// TIA Portal project "TFM_DanielBejar_S71500_Final" (V17)

(* hardware
DEVICE "S7-1500/ET200MP station_1"  S7-1500 station
   slot 0: "Rail_0"  Rack  6ES7 590-1***0-0AA0
   slot 0: "PS 25W 24VDC_1"  PS 25W 24VDC  6ES7 505-0KA00-0AB0  V1.0
   slot 1: "PLC_1"  CPU 1515-2 PN  6ES7 515-2AM02-0AB0  V2.9
      slot 3: "CPU display_1"  6ES7591-1BA00-0AA0
      slot 32768: "PROFINET interface_1"  X1
         slot 32769: "Port_1"  X1 P1
         slot 32770: "Port_2"  X1 P2
      slot 33024: "PROFINET interface_2"  X2
      slot 34817: "Virtual CP interface port_1"  Virtual CP interface port  Virtual CP interface port
   slot 2: "DI 32x24VDC BA_1"  DI 32x24VDC BA  6ES7 521-1BL10-0AA0  V1.1
   slot 3: "DQ 16x24VDC/0.5A BA_1"  DQ 16x24VDC/0.5A BA  6ES7 522-1BH10-0AA0  V1.1
DEVICE "HMI_1"  TP1200 Comfort
   slot 0: "HMI_1"  TP1200 Comfort  6AV2 124-0MC01-0AX0  17.0.0.0
   slot 1: "HMI_RT_1"  TP1200 Comfort  6AV2 124-0MC01-0AX0  17.0.0.0
   slot 5: "HMI_1.IE_CP_1"  PROFINET Interface  17.0.0.0
      slot 1: "PROFINET Interface_1"  PROFINET Interface
         slot 1: "Port_1"  Port
         slot 2: "Port_2"  Port
   slot 7: "HMI_1.MPI/DP_CP_1"  MPI/DP Interface  17.0.0.0
*)

// ===== PLC "PLC_1"  CPU 1515-2 PN =====

VAR_GLOBAL   // PLC tag table "Default tag table"
   "Clock_Byte" AT %MB255 : Byte;
   "Clock_10Hz" AT %M255.0 : Bool;
   "Clock_5Hz" AT %M255.1 : Bool;
   "Clock_2.5Hz" AT %M255.2 : Bool;
   "Clock_2Hz" AT %M255.3 : Bool;
   "Clock_1.25Hz" AT %M255.4 : Bool;
   "Clock_1Hz" AT %M255.5 : Bool;
   "Clock_0.625Hz" AT %M255.6 : Bool;
   "Clock_0.5Hz" AT %M255.7 : Bool;
END_VAR

VAR_GLOBAL   // PLC tag table "Estados"
   "Estado0" AT %M0.0 : Bool;
   "Estado1" AT %M0.1 : Bool;
   "Estado2" AT %M0.2 : Bool;
   "Estado3" AT %M0.3 : Bool;
   "Estado4" AT %M0.4 : Bool;
   "Estado5" AT %M0.5 : Bool;
   "Estado6" AT %M0.6 : Bool;
   "Estado7" AT %M0.7 : Bool;
   "Estado8" AT %M1.0 : Bool;
   "Estado9" AT %M1.1 : Bool;
   "Estado10" AT %M1.2 : Bool;
   "Estado11" AT %M1.3 : Bool;
   "Estado12" AT %M1.4 : Bool;
   "Estado13" AT %M1.5 : Bool;
   "EstadoPausa" AT %M1.6 : Bool;
   "EstadoError" AT %M1.7 : Bool;
   "Estados" AT %MD0 : DWord;
END_VAR

VAR_GLOBAL   // PLC tag table "IO_Programa"
   "SP_Cintas" AT %EW0 : Word;   // Cada bit se activará según los SP del final de las cintas de materiales
   "ActivacionCintas" AT %AW0 : Word;   // Cada bit indica la activación de una de las cintas
   "CintaGeneral" AT %A1.6 : Bool;   // Activación de la cinta general
   "SP_CintaGeneral" AT %E1.6 : Bool;   // Sensor de presencia de la cinta general
   "ReiniciarSistema" AT %E2.0 : Bool;   // Solicitud desde pulsador de reiniciar sistema
   "SP_CintaEmpaquetado" AT %E1.7 : Bool;   // Sensor de presencia de la cinta de empaquetado
   "CintaEmpaquetado" AT %A1.7 : Bool;   // Activación de la cinta de empaquetado
   "HMI_SP_Cintas" AT %MW10 : Word;   // Entrada simulada del HMI
   "HMI_SP_CintaGeneral" AT %M11.6 : Bool;   // Entrada simulada del HMI
   "HMI_SP_CintaEmpaquetado" AT %M11.7 : Bool;   // Entrada simulada del HMI
   "HMI_PaleE" AT %M12.0 : Bool;   // Entrada simulada del HMI
   "HMI_PaleF" AT %M12.1 : Bool;   // Entrada simulada del HMI
   "HMI_ReiniciarSistema" AT %M12.2 : Bool;   // Reiniciar el sistema desde HMI
END_VAR

DATA_BLOCK "TCP_vbes"   // DB6
{ S7_Optimized_Access := 'FALSE' }
VERSION : 0.1
   VAR
      RX : Array[0..49] of Char;   // Array del mensaje de entrada (RX)
      TX : Array[0..49] of Char;   // Array del mensaje de salida (TX)
      DesconectarServidor : Bool;   // Señal para desconectar el servidor
      TX_Enviar : Bool;   // Señal para enviar el mensaje en TX
      TX_Procesando : Bool;   // Hasta no recibir el ACK, esta vbe será true
      RX_Recibir : Bool := true;   // Habilita la recepción de mensajes
      RX_Procesar : Bool;   // Cuando se recibe un mensaje, se manda a procesar
      TX_Len : UDInt;   // Longitud mensaje TX
      RX_Len : UDInt;   // Longitud mensaje RX
      LastID : Char;   // Ultimo mensaje mandado (para comprobar el ACK)
      TiempoTX : Time;   // Tiempo del sistema cuando se mandó el último TX
      TiempoRX : Time;   // Tiempo del sistema cuando se recibió el último RX
   END_VAR
BEGIN
END_DATA_BLOCK

DATA_BLOCK "SISTEMA_vbes"   // DB8
{ S7_Optimized_Access := 'FALSE' }
VERSION : 0.1
   VAR
      Mesa : Array[0..15] of Word;   // Los bits de Mesa indican si el componente está presente o no en la posición de esa mesa
      Prioridad : Array[0..15] of Int;   // A menor sea el índice, mayor prioridad tiene dicha mesa. Almacena el número de mesa
      Material_Destino : Word;   // Material que será transportado por la cinta general
      Mesa_Destino : Int;   // Mesa en la que irá el material que circula por la cinta general
      Material_EnProceso : Word;   // Variable temporal que almacena el material que el robot está colocando
      Mesa_EnProceso : Int;   // Variable temporal que almacena la mesa que el robot está utilizando
      Mascaras_Cintas : Word;   // Deshabilita un SP de la cinta de materiales. Ocurre cuando el material no es necesario
      NumeroMesas : Word := 4;   // Número de mesas reales en el sistema (máximo 16)
      SP_Enmascarados : Word;   // Los sensores de presencia tras tener en cuenta cuáles están deshabilitados
      IndicePrioridad : Int;   // Indice de la matriz de prioridades
      MatsNecesarios : Word;   // Inversa del contenido en Mesa[]
      SP_Prioritarios : Word;   // Los bits de esta vbe indican si el alimento está disponible y es necesario para la mesa prioritaria
      NumeroMateriales : Int := 5;   // Numero de materiales sin contar caja y tapa
      RobotOcupado : Bool;   // True si el robot está realizando alguna operación
      RobotConectado : Bool;   // True si la conexión con el robot es correcta
      MsgError : String;   // Almacena el último mensaje que ha causado un error
      ElementoBase : Word := 16#20;   // El identificador de la base es bit(NumMateriales)
      ElementoTapa : Word := 16#40;   // El identificador de la tapa es bit(NumMateriales+1)
      ModoSimulacion : Bool;   // Determina si el modo simulación está activo o no
      TActivacionCintaEmp : Time;   // Tiempo hasta el que debe mantenerse activa la cinta de empaquetado
      EstadoAnterior : Word;   // Almacena el estado anterior, sirve para retomar el funcionamiento tras un fallo leve
   END_VAR
BEGIN
   Prioridad[0] := 0;
   Prioridad[1] := 1;
   Prioridad[2] := 2;
   Prioridad[3] := 3;
   Prioridad[4] := 4;
   Prioridad[5] := 5;
   Prioridad[6] := 6;
   Prioridad[7] := 7;
   Prioridad[8] := 8;
   Prioridad[9] := 9;
   Prioridad[10] := 10;
   Prioridad[11] := 11;
   Prioridad[12] := 12;
   Prioridad[13] := 13;
   Prioridad[14] := 14;
   Prioridad[15] := 15;
END_DATA_BLOCK

DATA_BLOCK "HMI_vbes"   // DB9
{ S7_Optimized_Access := 'FALSE' }
VERSION : 0.1
   VAR
      HMI_NumeroMesaSeleccionada : Int;
      HMI_ValorMesaSeleccionada : Word;
      HMI_MesaSeleccionada : Bool;
      HMI_BaseSeleccionada : Bool;
      HMI_TapaSeleccionada : Bool;
      HMI_NumeroMesasDeseadas : Int := 4;
      HMI_NumeroMaterialesDeseados : Int := 5;
      HMI_MostrarPiezaE : Bool;
      HMI_MostrarPiezaF : Bool;
      HMI_MaterialDestino : Word;
      HMI_MesaDestino : Word;
      HMI_Errores : Word;
      HMI_MandarHome : Bool;
      HMI_ApagarRobot : Bool;
      HMI_PausarSistema : Bool;
      HMI_SistemaPausado : Bool;
   END_VAR
BEGIN
END_DATA_BLOCK

// folder: System blocks/Program resources

DATA_BLOCK "TCP_COMMS_DB"   // DB1
{ S7_Optimized_Access := 'TRUE' }
VERSION : 0.1
// stored: InstanceOfName TCP_COMMS
"TCP_COMMS"
BEGIN
END_DATA_BLOCK

DATA_BLOCK "DB_ParamsConexion"   // DB2
{ S7_Optimized_Access := 'TRUE' }
AUTHOR : SIMATIC
FAMILY : MC7Plus
NAME : TC_IP_v4
VERSION : 1.0
// stored: InstanceOfName TCON_IP_v4
"TCON_IP_v4"
BEGIN
   ID := 1;
   InterfaceId := 64;
   RemotePort := 2000;
   ActiveEstablished := true;
   RemoteAddress.ADDR[1] := 192;
   RemoteAddress.ADDR[2] := 168;
   RemoteAddress.ADDR[4] := 130;
END_DATA_BLOCK

// folder: (top level)

FUNCTION_BLOCK "TCP_COMMS"   // FB1, LAD
TITLE = Bloque de comunicaciones TCP
{ S7_Optimized_Access := 'TRUE' }
VERSION : 0.1
// Este bloque está encargado de conectar, desconectar, enviar y recibir mensajes por el puerto TCP. El PLC trabaja como cliente. Los datos necesarios para este bloque se encuentran en TCP_DATA.
   VAR
      TCON : Struct
         REQ : Bool;
         DONE : Bool;
         BUSY : Bool;
         ERROR : Bool;
         STATUS : UInt;
         CONNECTED : Bool;
      END_STRUCT;
      TDISCON : Struct
         REQ : Bool;
         DONE : Bool;
         BUSY : Bool;
         ERROR : Bool;
         STATUS : UInt;
      END_STRUCT;
      TSEND : Struct
         REQ : Bool;
         DONE : Bool;
         BUSY : Bool;
         ERROR : Bool;
         STATUS : UInt;
      END_STRUCT;
      TRCV : Struct
         EN_R : Bool;
         NDR : Bool;
         BUSY : Bool;
         ERROR : Bool;
         STATUS : UInt;
         RCVD_LEN : UInt;
      END_STRUCT;
      IntentosTX : Int;
   END_VAR
   VAR CONSTANT
      MaxIntentosTX : Int := 10;
   END_VAR
   VAR_TEMP   // added for the SCL form of the ladder/FBD networks
      _w1 : Bool;
      _w2 : Bool;
   END_VAR
BEGIN

REGION Network 1: Conexión con el servidor TCP
   // Si se habilita, permite la conexión del PLC con el server.
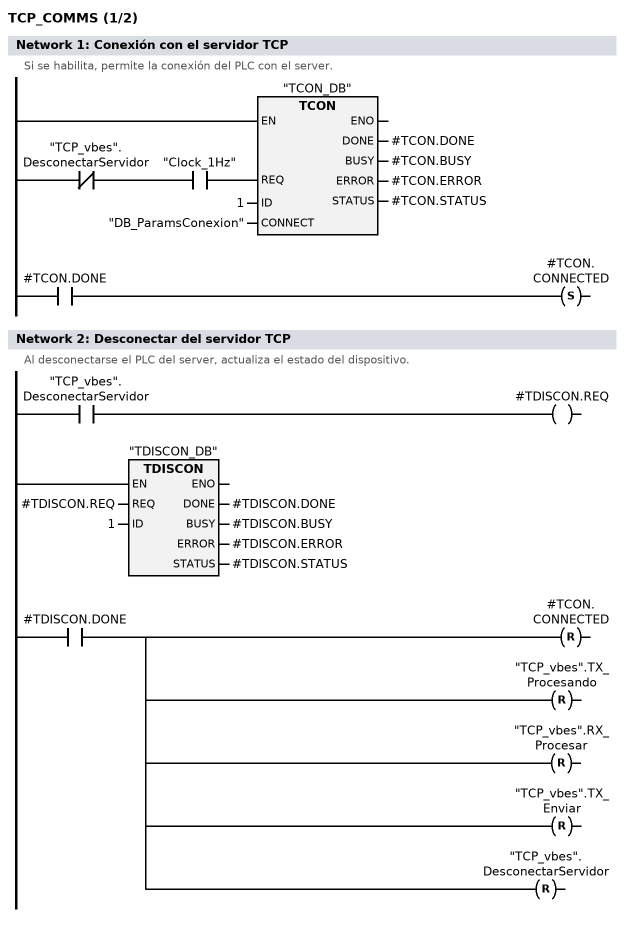
   "TCON_DB"(REQ := NOT "TCP_vbes".DesconectarServidor AND "Clock_1Hz",   // TCON
             ID := 1,
             CONNECT := "DB_ParamsConexion",
             DONE => #TCON.DONE,
             BUSY => #TCON.BUSY,
             ERROR => #TCON.ERROR,
             STATUS => #TCON.STATUS);
   IF #TCON.DONE THEN #TCON.CONNECTED := TRUE; END_IF;
END_REGION

REGION Network 2: Desconectar del servidor TCP
   // Al desconectarse el PLC del server, actualiza el estado del dispositivo.
   #TDISCON.REQ := "TCP_vbes".DesconectarServidor;
   "TDISCON_DB"(REQ := #TDISCON.REQ,   // TDISCON
                ID := 1,
                DONE => #TDISCON.DONE,
                BUSY => #TDISCON.BUSY,
                ERROR => #TDISCON.ERROR,
                STATUS => #TDISCON.STATUS);
   IF #TDISCON.DONE THEN
       #TCON.CONNECTED := FALSE;
       "TCP_vbes".TX_Procesando := FALSE;
       "TCP_vbes".RX_Procesar := FALSE;
       "TCP_vbes".TX_Enviar := FALSE;
       "TCP_vbes".DesconectarServidor := FALSE;
   END_IF;
END_REGION

REGION Network 3: Transmitir datos hacia el servidor (TX)
   // Si hay datos que enviar, el sistema está conectado y no se está procesando una escritura anterior, se manda el buffer TX.
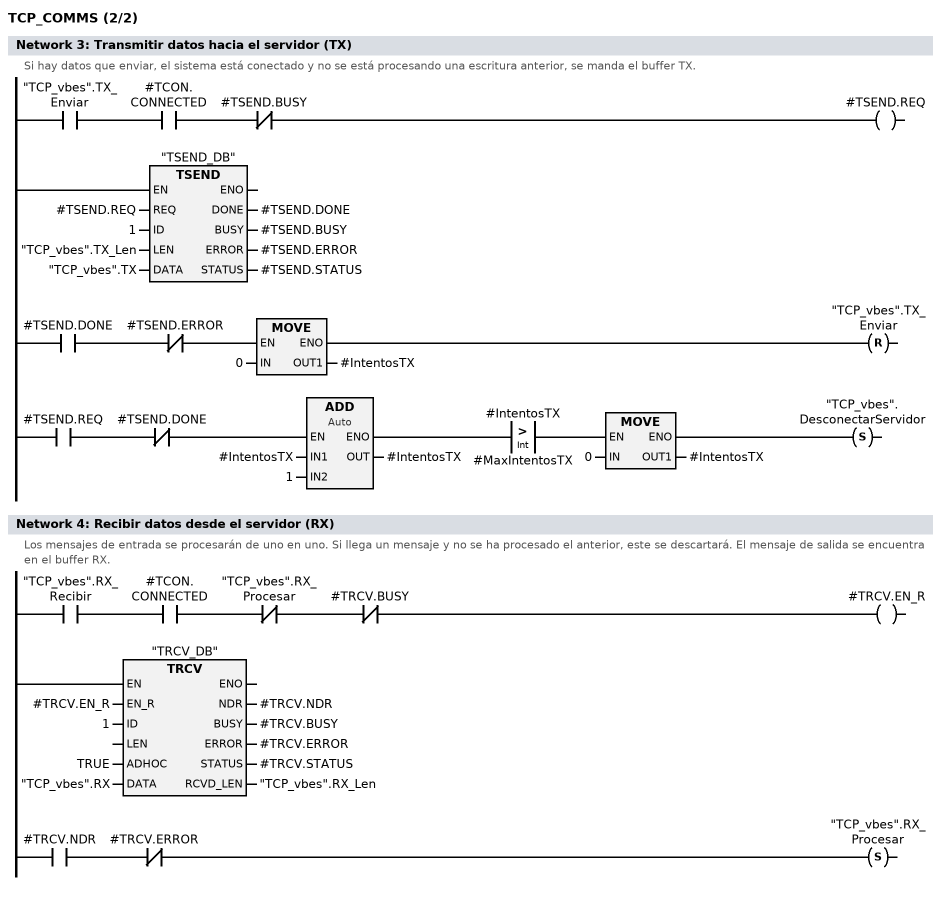
   #TSEND.REQ := "TCP_vbes".TX_Enviar AND #TCON.CONNECTED AND NOT #TSEND.BUSY;
   "TSEND_DB"(REQ := #TSEND.REQ,   // TSEND
              ID := 1,
              LEN := "TCP_vbes".TX_Len,
              DATA := "TCP_vbes".TX,
              DONE => #TSEND.DONE,
              BUSY => #TSEND.BUSY,
              ERROR => #TSEND.ERROR,
              STATUS => #TSEND.STATUS);
   IF #TSEND.DONE AND NOT #TSEND.ERROR THEN
       #IntentosTX := 0;
       "TCP_vbes".TX_Enviar := FALSE;
   END_IF;
   #_w1 := #TSEND.REQ AND NOT #TSEND.DONE;
   IF #_w1 THEN #IntentosTX := #IntentosTX + 1; END_IF;
   #_w2 := #_w1 AND (#IntentosTX > #MaxIntentosTX);
   IF #_w2 THEN
       #IntentosTX := 0;
       "TCP_vbes".DesconectarServidor := TRUE;
   END_IF;
END_REGION

REGION Network 4: Recibir datos desde el servidor (RX)
   // Los mensajes de entrada se procesarán de uno en uno. Si llega un mensaje y no se ha procesado el anterior, este se descartará. El mensaje de salida se encuentra en el buffer RX.
   #TRCV.EN_R := "TCP_vbes".RX_Recibir AND #TCON.CONNECTED AND NOT "TCP_vbes".RX_Procesar AND NOT #TRCV.BUSY;
   "TRCV_DB"(EN_R := #TRCV.EN_R,   // TRCV
             ID := 1,
             ADHOC := TRUE,
             DATA := "TCP_vbes".RX,
             NDR => #TRCV.NDR,
             BUSY => #TRCV.BUSY,
             ERROR => #TRCV.ERROR,
             STATUS => #TRCV.STATUS,
             RCVD_LEN => "TCP_vbes".RX_Len);
   IF #TRCV.NDR AND NOT #TRCV.ERROR THEN "TCP_vbes".RX_Procesar := TRUE; END_IF;
END_REGION
END_FUNCTION_BLOCK

FUNCTION "SeleccionarMateriales" : Void   // FC1, LAD
TITLE = Selección de materiales
{ S7_Optimized_Access := 'TRUE' }
VERSION : 0.1
   VAR_TEMP
      AuxVar : Word;   // Word auxiliar
      TX_Realizado : Bool;   // True si el TX se ha realizado correctamente
      SimSP_Cintas : Word;   // OR de las entradas reales y simuladas
      SimSP_CintaGeneral : Bool;   // OR de los sensores reales y simulados de la cinta general
      SimSP_CintaEmpaq : Bool;   // OR de los sensores reales y simulados de cinta empaquetadora
      TiempoAux : Time;   // Time auxiliar
   END_VAR
   VAR_TEMP   // added for the SCL form of the ladder/FBD networks
      _w1 : Bool;
      _w2 : Bool;
      _w3 : Bool;
      _w4 : Bool;
      _w5 : Bool;
      _w6 : Bool;
   END_VAR
BEGIN

REGION Network 1: Genera las entradas simuladas de estar en el modo de simulación
   // Se unen las entradas HMI con las entradas digitales del sistema en el modo de simulación.
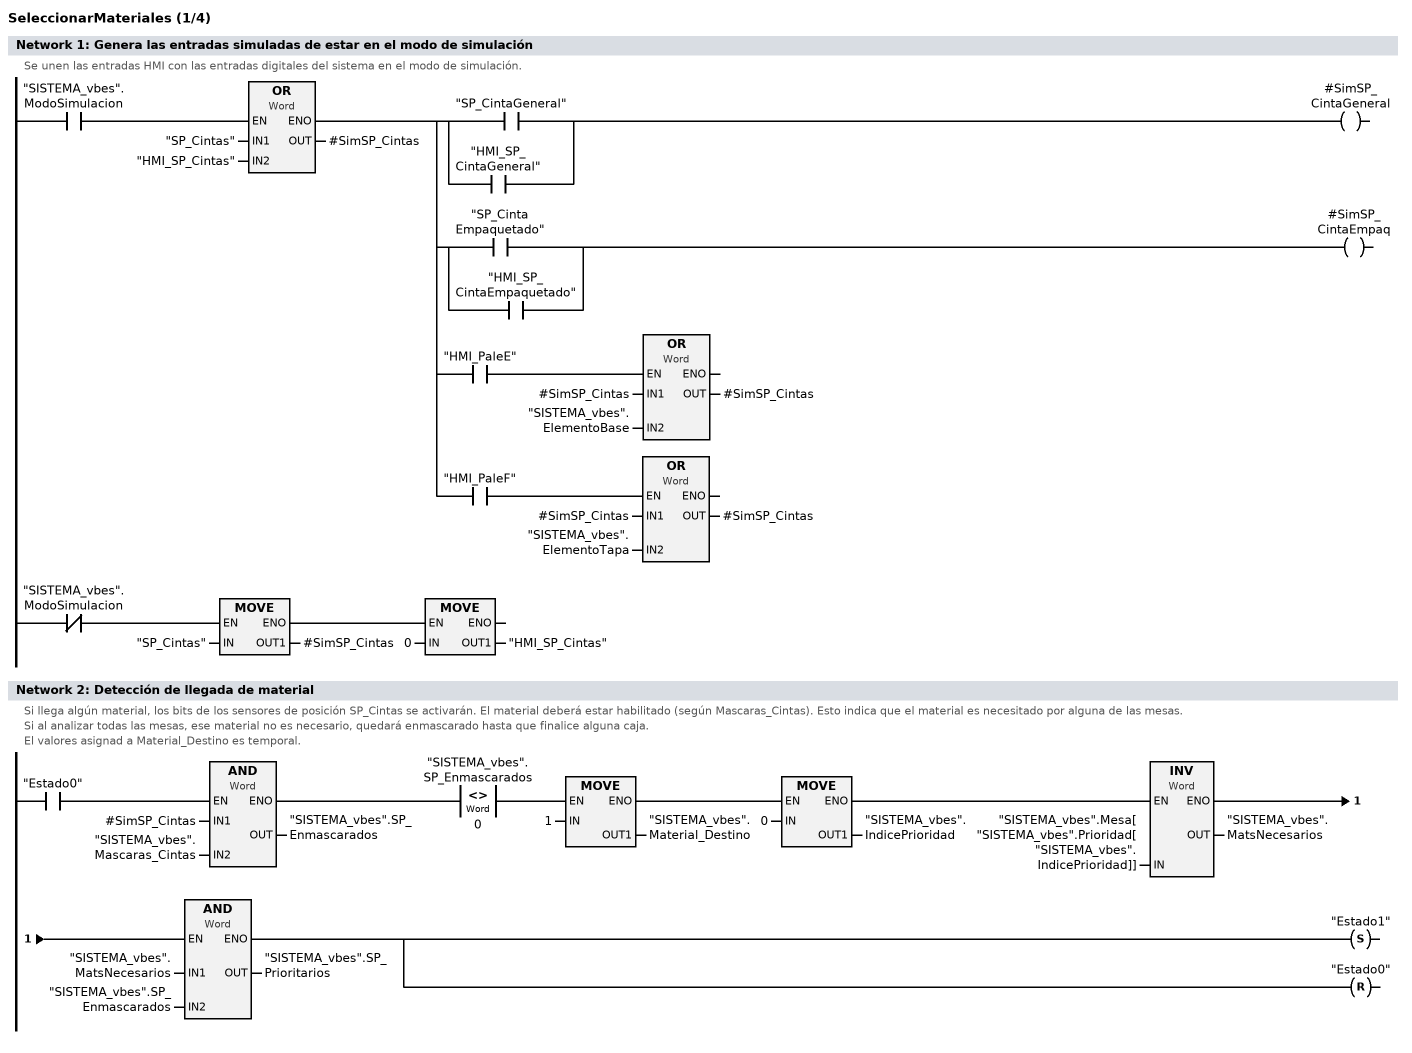
   IF "SISTEMA_vbes".ModoSimulacion THEN #SimSP_Cintas := "SP_Cintas" OR "HMI_SP_Cintas"; END_IF;
   #SimSP_CintaGeneral := "SISTEMA_vbes".ModoSimulacion AND ("SP_CintaGeneral" OR "HMI_SP_CintaGeneral");
   #SimSP_CintaEmpaq := "SISTEMA_vbes".ModoSimulacion AND ("SP_CintaEmpaquetado" OR "HMI_SP_CintaEmpaquetado");
   IF "SISTEMA_vbes".ModoSimulacion AND "HMI_PaleE" THEN
       #SimSP_Cintas := #SimSP_Cintas OR "SISTEMA_vbes".ElementoBase;
   END_IF;
   IF "SISTEMA_vbes".ModoSimulacion AND "HMI_PaleF" THEN
       #SimSP_Cintas := #SimSP_Cintas OR "SISTEMA_vbes".ElementoTapa;
   END_IF;
   IF NOT "SISTEMA_vbes".ModoSimulacion THEN
       #SimSP_Cintas := "SP_Cintas";
       "HMI_SP_Cintas" := 0;
   END_IF;
END_REGION

REGION Network 2: Detección de llegada de material
   // Si llega algún material, los bits de los sensores de posición SP_Cintas se activarán. El material deberá estar habilitado (según Mascaras_Cintas). Esto indica que el material es necesitado por alguna de las mesas.
   // Si al analizar todas las mesas, ese material no es necesario, quedará enmascarado hasta que finalice alguna caja.
   // El valores asignad a Material_Destino es temporal.
   RUNG wire#powerrail
      Contact( "Estado0" )
      { S7_Templates := "SrcType := Word" } And(in1 := #SimSP_Cintas, in2 := "SISTEMA_vbes".Mascaras_Cintas, out => "SISTEMA_vbes".SP_Enmascarados)
      { S7_Templates := "SrcType := Word" } NE_Contact(in1 := "SISTEMA_vbes".SP_Enmascarados, in2 := 0)
      Move(in := 1, out1 => "SISTEMA_vbes".Material_Destino)
      Move(in := 0, out1 => "SISTEMA_vbes".IndicePrioridad)
      { S7_Templates := "SrcType := Word" } Inv(in := "SISTEMA_vbes".Mesa["SISTEMA_vbes".Prioridad["SISTEMA_vbes".IndicePrioridad]], out => "SISTEMA_vbes".MatsNecesarios)
      { S7_Templates := "SrcType := Word" } And(in1 := "SISTEMA_vbes".MatsNecesarios, in2 := "SISTEMA_vbes".SP_Enmascarados, out => "SISTEMA_vbes".SP_Prioritarios)
      wire#w1
      S_Coil( "Estado1" )
   END_RUNG
   RUNG wire#w1
      R_Coil( "Estado0" )
   END_RUNG
   // the same network as SCL:
   IF "Estado0" THEN
       "SISTEMA_vbes".SP_Enmascarados := #SimSP_Cintas AND "SISTEMA_vbes".Mascaras_Cintas;
   END_IF;
   IF "Estado0" AND ("SISTEMA_vbes".SP_Enmascarados <> 0) THEN
       "SISTEMA_vbes".Material_Destino := 1;
       "SISTEMA_vbes".IndicePrioridad := 0;
       "SISTEMA_vbes".MatsNecesarios := NOT "SISTEMA_vbes".Mesa["SISTEMA_vbes".Prioridad["SISTEMA_vbes".IndicePrioridad]];
       "SISTEMA_vbes".SP_Prioritarios := "SISTEMA_vbes".MatsNecesarios AND "SISTEMA_vbes".SP_Enmascarados;
       "Estado1" := TRUE;
       "Estado0" := FALSE;
   END_IF;
END_REGION

REGION Network 3: Selección de un solo material según mesa prioritaria
   // Si por lo que fuera llegase más de un material, habría que elegir uno solo que comprobar. Habrá que seleccionar además aquél material que necesiten las mesas en orden de prioridad.
   // Aquí se itera dentro del array Prioridad[] mediante el índice IndicePrioridad. El máximo de mesas queda definido por NumeroMesas.
   // 
   // Si el índice supera el número de mesas indica que los materiales que habían por procesar y que han disparado los SP NO son necesarios hasta que se liberen alguna de las cajas, por lo 
   // tanto, se deshabilitan todos los materiales que hayan disparado el SP.
   // 
   // La variable SP_Prioritarios almacena aquellos componentes que la Mesa[IndicePrioridad] necesita Y que están dentro de las cintas. Si es distinto de cero, indica que hay un material dentro 
   // de las cintas que es necesario para la mesa. Únicamente falta encontrar qué material es; es decir, en qué posición de SP_Prioritarios se encuentra.
   // 
   // La función AND (SP_Prioritarios  AND 1) comprueba que el LSB es 1 o 0. Si es uno, ya se ha encontrado el material y por lo tanto, se actualiza el valor de Mesa_Destino, deja activada la cinta
   // correspondiente a ese material y cambia de estado. Antes de hacer esto, se debe comprobar si ya hay una bandeja en la mesa que se dispone a colocar.
   // 
   // Si el valor es cero, hay que pasar al siguiente Material_Destino (son potencias de 2, luego bitshift a la izquierda) y pasar a comprobar el siguiente bit  de SP_Prioritarios haciendo un bitshift
   // a la derecha.
   // 
   // Cuando SP_Prioritarios es 0, indica que NO queda ningún material que sea necesario para esa Mesa[IndicePrioridad], por lo tanto, se incrementa el contador IndicePrioridad y se vuelve a calcular 
   // SP_Prioritarios pero para la nueva mesa.
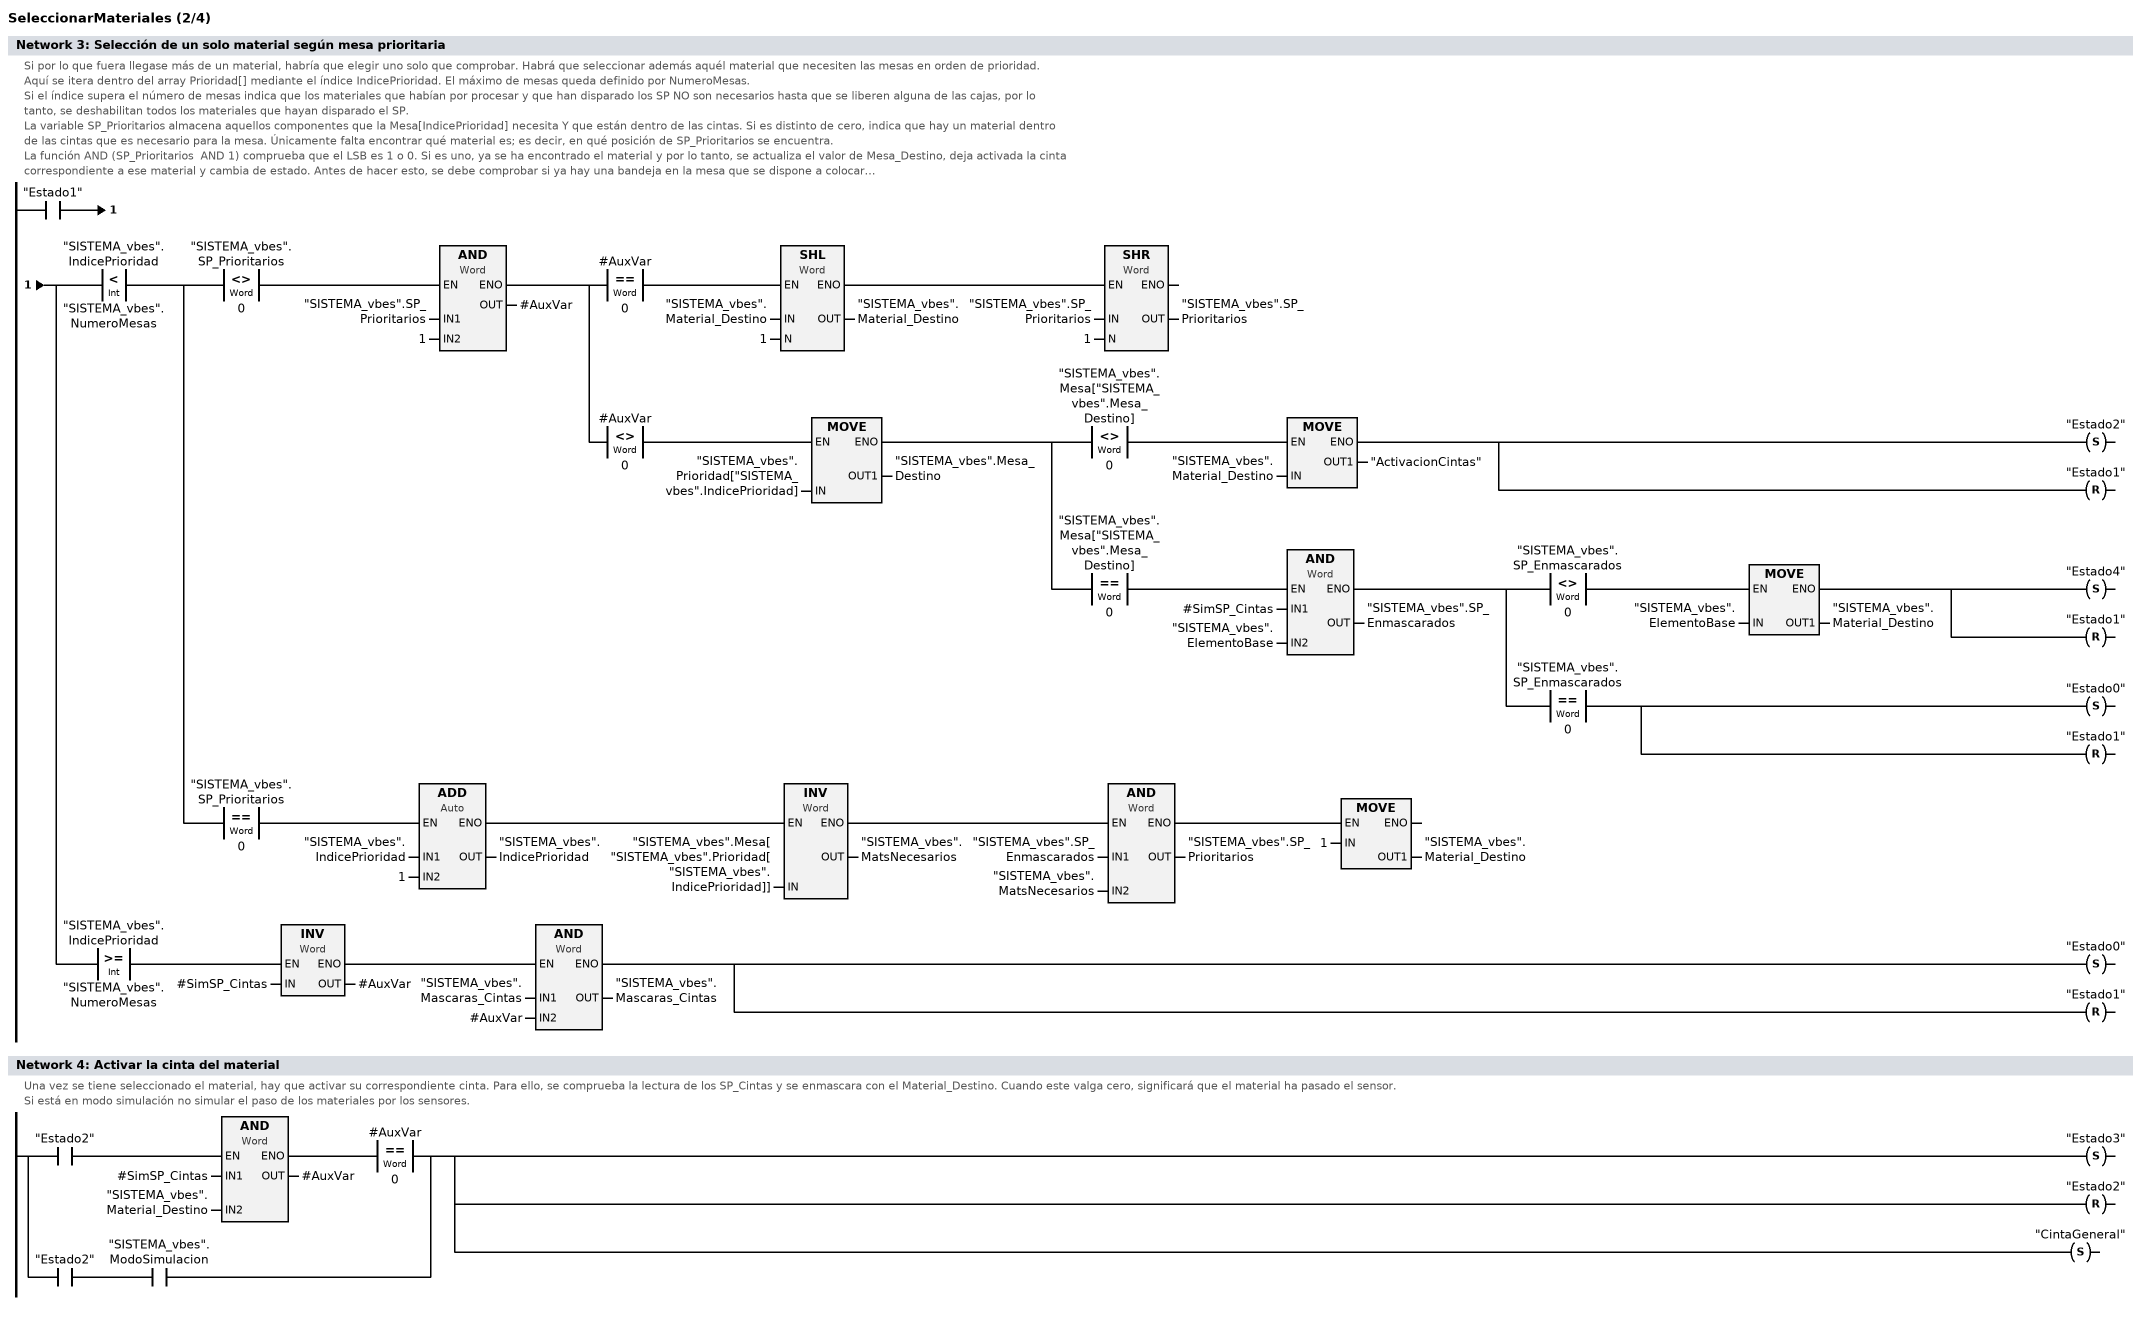
   RUNG wire#powerrail
      Contact( "Estado1" )
      wire#w1
      { S7_Templates := "SrcType := Int" } LT_Contact(in1 := "SISTEMA_vbes".IndicePrioridad, in2 := "SISTEMA_vbes".NumeroMesas)
      wire#w2
      { S7_Templates := "SrcType := Word" } NE_Contact(in1 := "SISTEMA_vbes".SP_Prioritarios, in2 := 0)
      { S7_Templates := "SrcType := Word" } And(in1 := "SISTEMA_vbes".SP_Prioritarios, in2 := 1, out => #AuxVar)
      wire#w3
      { S7_Templates := "SrcType := Word" } EQ_Contact(in1 := #AuxVar, in2 := 0)
      { S7_Templates := "SrcType := Word" } Shl(in := "SISTEMA_vbes".Material_Destino, n := 1, out => "SISTEMA_vbes".Material_Destino)
      { S7_Templates := "SrcType := Word" } Shr(in := "SISTEMA_vbes".SP_Prioritarios, n := 1, out => "SISTEMA_vbes".SP_Prioritarios)
   END_RUNG
   RUNG wire#w3
      { S7_Templates := "SrcType := Word" } NE_Contact(in1 := #AuxVar, in2 := 0)
      Move(in := "SISTEMA_vbes".Prioridad["SISTEMA_vbes".IndicePrioridad], out1 => "SISTEMA_vbes".Mesa_Destino)
      wire#w4
      { S7_Templates := "SrcType := Word" } NE_Contact(in1 := "SISTEMA_vbes".Mesa["SISTEMA_vbes".Mesa_Destino], in2 := 0)
      Move(in := "SISTEMA_vbes".Material_Destino, out1 => "ActivacionCintas")
      wire#w5
      S_Coil( "Estado2" )
   END_RUNG
   RUNG wire#w5
      R_Coil( "Estado1" )
   END_RUNG
   RUNG wire#w4
      { S7_Templates := "SrcType := Word" } EQ_Contact(in1 := "SISTEMA_vbes".Mesa["SISTEMA_vbes".Mesa_Destino], in2 := 0)
      { S7_Templates := "SrcType := Word" } And(in1 := #SimSP_Cintas, in2 := "SISTEMA_vbes".ElementoBase, out => "SISTEMA_vbes".SP_Enmascarados)
      wire#w6
      { S7_Templates := "SrcType := Word" } NE_Contact(in1 := "SISTEMA_vbes".SP_Enmascarados, in2 := 0)
      Move(in := "SISTEMA_vbes".ElementoBase, out1 => "SISTEMA_vbes".Material_Destino)
      wire#w7
      S_Coil( "Estado4" )
   END_RUNG
   RUNG wire#w7
      R_Coil( "Estado1" )
   END_RUNG
   RUNG wire#w6
      { S7_Templates := "SrcType := Word" } EQ_Contact(in1 := "SISTEMA_vbes".SP_Enmascarados, in2 := 0)
      wire#w8
      S_Coil( "Estado0" )
   END_RUNG
   RUNG wire#w8
      R_Coil( "Estado1" )
   END_RUNG
   RUNG wire#w2
      { S7_Templates := "SrcType := Word" } EQ_Contact(in1 := "SISTEMA_vbes".SP_Prioritarios, in2 := 0)
      Add(in1 := "SISTEMA_vbes".IndicePrioridad, in2 := 1, out => "SISTEMA_vbes".IndicePrioridad)
      { S7_Templates := "SrcType := Word" } Inv(in := "SISTEMA_vbes".Mesa["SISTEMA_vbes".Prioridad["SISTEMA_vbes".IndicePrioridad]], out => "SISTEMA_vbes".MatsNecesarios)
      { S7_Templates := "SrcType := Word" } And(in1 := "SISTEMA_vbes".SP_Enmascarados, in2 := "SISTEMA_vbes".MatsNecesarios, out => "SISTEMA_vbes".SP_Prioritarios)
      Move(in := 1, out1 => "SISTEMA_vbes".Material_Destino)
   END_RUNG
   RUNG wire#w1
      { S7_Templates := "SrcType := Int" } GE_Contact(in1 := "SISTEMA_vbes".IndicePrioridad, in2 := "SISTEMA_vbes".NumeroMesas)
      { S7_Templates := "SrcType := Word" } Inv(in := #SimSP_Cintas, out => #AuxVar)
      { S7_Templates := "SrcType := Word" } And(in1 := "SISTEMA_vbes".Mascaras_Cintas, in2 := #AuxVar, out => "SISTEMA_vbes".Mascaras_Cintas)
      wire#w9
      S_Coil( "Estado0" )
   END_RUNG
   RUNG wire#w9
      R_Coil( "Estado1" )
   END_RUNG
   // the same network as SCL:
   #_w1 := "Estado1" AND ("SISTEMA_vbes".IndicePrioridad < "SISTEMA_vbes".NumeroMesas);
   #_w2 := #_w1 AND ("SISTEMA_vbes".SP_Prioritarios <> 0);
   IF #_w2 THEN #AuxVar := "SISTEMA_vbes".SP_Prioritarios AND 1; END_IF;
   IF #_w2 AND (#AuxVar = 0) THEN
       "SISTEMA_vbes".Material_Destino := SHL(IN := "SISTEMA_vbes".Material_Destino, N := 1);
       "SISTEMA_vbes".SP_Prioritarios := SHR(IN := "SISTEMA_vbes".SP_Prioritarios, N := 1);
   END_IF;
   #_w3 := #_w2 AND (#AuxVar <> 0);
   IF #_w3 THEN
       "SISTEMA_vbes".Mesa_Destino := "SISTEMA_vbes".Prioridad["SISTEMA_vbes".IndicePrioridad];
   END_IF;
   IF #_w3 AND ("SISTEMA_vbes".Mesa["SISTEMA_vbes".Mesa_Destino] <> 0) THEN
       "ActivacionCintas" := "SISTEMA_vbes".Material_Destino;
       "Estado2" := TRUE;
   END_IF;
   #_w4 := "Estado1";
   IF #_w3 AND ("SISTEMA_vbes".Mesa["SISTEMA_vbes".Mesa_Destino] <> 0) THEN "Estado1" := FALSE; END_IF;
   #_w5 := #_w3 AND ("SISTEMA_vbes".Mesa["SISTEMA_vbes".Mesa_Destino] = 0);
   IF #_w5 THEN "SISTEMA_vbes".SP_Enmascarados := #SimSP_Cintas AND "SISTEMA_vbes".ElementoBase; END_IF;
   IF #_w5 AND ("SISTEMA_vbes".SP_Enmascarados <> 0) THEN
       "SISTEMA_vbes".Material_Destino := "SISTEMA_vbes".ElementoBase;
       "Estado4" := TRUE;
       "Estado1" := FALSE;
   END_IF;
   IF #_w5 AND ("SISTEMA_vbes".SP_Enmascarados = 0) THEN
       "Estado0" := TRUE;
       "Estado1" := FALSE;
   END_IF;
   IF #_w1 AND ("SISTEMA_vbes".SP_Prioritarios = 0) THEN
       "SISTEMA_vbes".IndicePrioridad := "SISTEMA_vbes".IndicePrioridad + 1;
       "SISTEMA_vbes".MatsNecesarios := NOT "SISTEMA_vbes".Mesa["SISTEMA_vbes".Prioridad["SISTEMA_vbes".IndicePrioridad]];
   END_IF;
   #_w6 := #_w1 AND ("SISTEMA_vbes".SP_Prioritarios = 0);
   IF #_w6 THEN
       "SISTEMA_vbes".SP_Prioritarios := "SISTEMA_vbes".SP_Enmascarados AND "SISTEMA_vbes".MatsNecesarios;
       "SISTEMA_vbes".Material_Destino := 1;
   END_IF;
   IF #_w4 AND ("SISTEMA_vbes".IndicePrioridad >= "SISTEMA_vbes".NumeroMesas) THEN
       #AuxVar := NOT #SimSP_Cintas;
       "SISTEMA_vbes".Mascaras_Cintas := "SISTEMA_vbes".Mascaras_Cintas AND #AuxVar;
       "Estado0" := TRUE;
       "Estado1" := FALSE;
   END_IF;
END_REGION

REGION Network 4: Activar la cinta del material
   // Una vez se tiene seleccionado el material, hay que activar su correspondiente cinta. Para ello, se comprueba la lectura de los SP_Cintas y se enmascara con el Material_Destino. Cuando este valga cero, significará que el material ha pasado el sensor.
   // Si está en modo simulación no simular el paso de los materiales por los sensores.
   RUNG wire#powerrail
      Contact( "Estado2" )
      { S7_Templates := "SrcType := Word" } And(in1 := #SimSP_Cintas, in2 := "SISTEMA_vbes".Material_Destino, out => #AuxVar)
      { S7_Templates := "SrcType := Word" } EQ_Contact(in1 := #AuxVar, in2 := 0)
      wire#w1
      S_Coil( "Estado3" )
   END_RUNG
   RUNG wire#powerrail
      Contact( "Estado2" )
      Contact( "SISTEMA_vbes".ModoSimulacion )
   END_RUNG wire#w1
   RUNG wire#w1
      R_Coil( "Estado2" )
   END_RUNG
   RUNG wire#w1
      S_Coil( "CintaGeneral" )
   END_RUNG
   // the same network as SCL:
   IF "Estado2" THEN #AuxVar := #SimSP_Cintas AND "SISTEMA_vbes".Material_Destino; END_IF;
   IF ("Estado2" AND (#AuxVar = 0)) OR ("Estado2" AND "SISTEMA_vbes".ModoSimulacion) THEN
       "Estado3" := TRUE;
   END_IF;
   #_w1 := ("Estado2" AND (#AuxVar = 0)) OR ("Estado2" AND "SISTEMA_vbes".ModoSimulacion);
   IF #_w1 THEN
       "Estado2" := FALSE;
       "CintaGeneral" := TRUE;
   END_IF;
END_REGION

REGION Network 5: Activar la cinta general
   // La cinta general alcanza el material al brazo robótico.
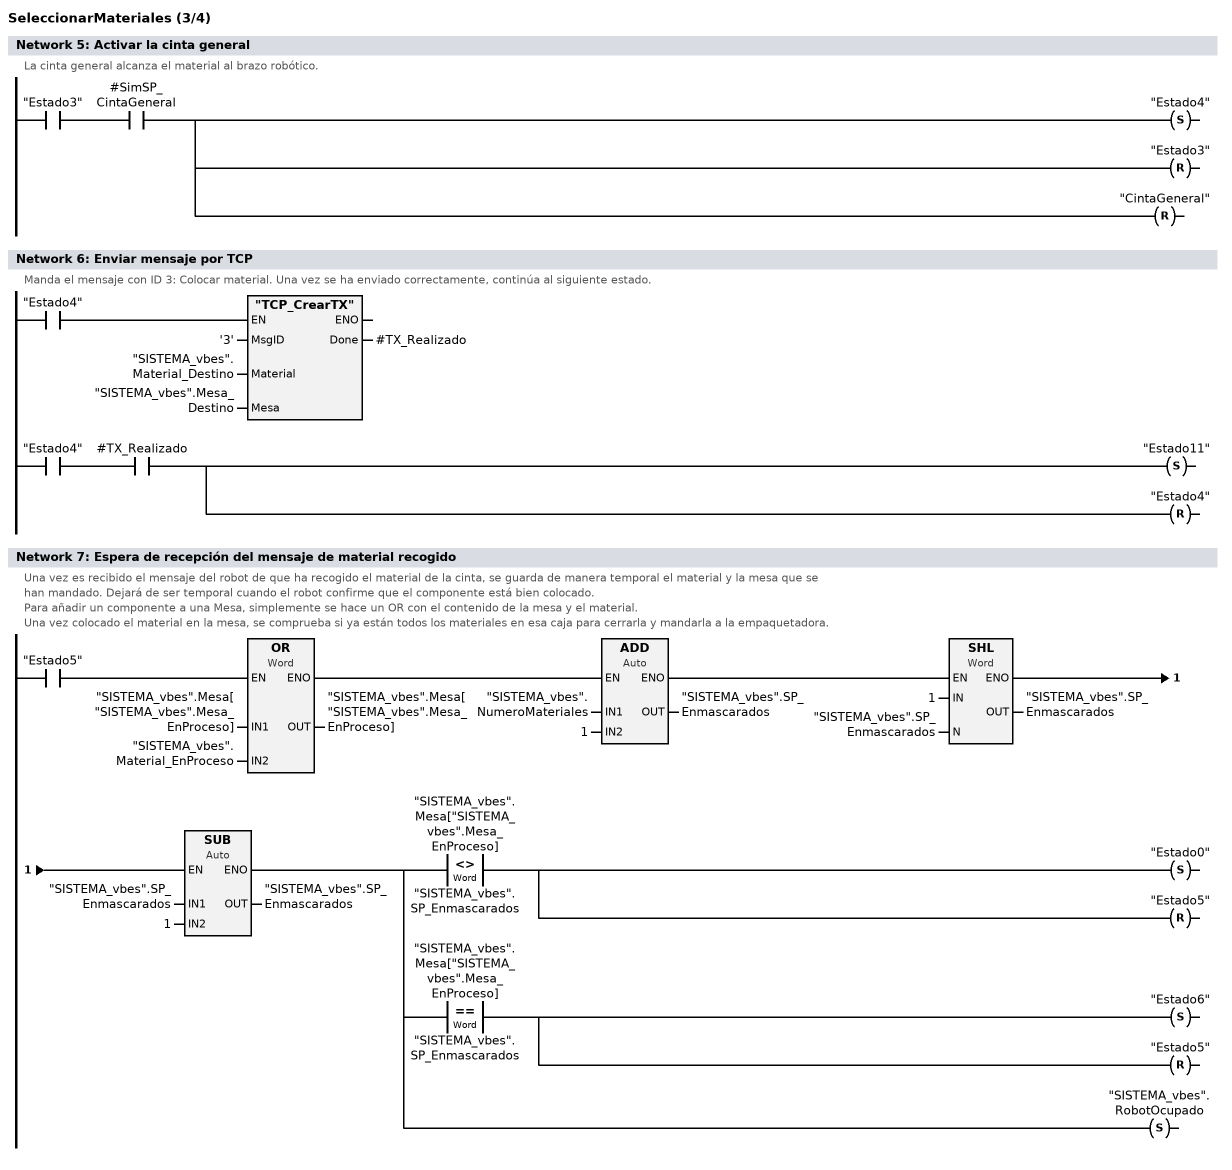
   RUNG wire#powerrail
      Contact( "Estado3" )
      Contact( #SimSP_CintaGeneral )
      wire#w1
      S_Coil( "Estado4" )
   END_RUNG
   RUNG wire#w1
      R_Coil( "Estado3" )
   END_RUNG
   RUNG wire#w1
      R_Coil( "CintaGeneral" )
   END_RUNG
   // the same network as SCL:
   IF "Estado3" AND #SimSP_CintaGeneral THEN "Estado4" := TRUE; END_IF;
   #_w1 := "Estado3" AND #SimSP_CintaGeneral;
   IF #_w1 THEN
       "Estado3" := FALSE;
       "CintaGeneral" := FALSE;
   END_IF;
END_REGION

REGION Network 6: Enviar mensaje por TCP
   // Manda el mensaje con ID 3: Colocar material. Una vez se ha enviado correctamente, continúa al siguiente estado.
   RUNG wire#powerrail
      Contact( "Estado4" )
      "TCP_CrearTX"(MsgID := '3', Material := "SISTEMA_vbes".Material_Destino, Mesa := "SISTEMA_vbes".Mesa_Destino, Done => #TX_Realizado)
   END_RUNG
   RUNG wire#powerrail
      Contact( "Estado4" )
      Contact( #TX_Realizado )
      wire#w1
      S_Coil( "Estado11" )
   END_RUNG
   RUNG wire#w1
      R_Coil( "Estado4" )
   END_RUNG
   // the same network as SCL:
   IF "Estado4" THEN
       "TCP_CrearTX"(MsgID := '3',
                     Material := "SISTEMA_vbes".Material_Destino,
                     Mesa := "SISTEMA_vbes".Mesa_Destino,
                     Done => #TX_Realizado);
   END_IF;
   IF "Estado4" AND #TX_Realizado THEN
       "Estado11" := TRUE;
       "Estado4" := FALSE;
   END_IF;
END_REGION

REGION Network 7: Espera de recepción del mensaje de material recogido
   // Una vez es recibido el mensaje del robot de que ha recogido el material de la cinta, se guarda de manera temporal el material y la mesa que se 
   // han mandado. Dejará de ser temporal cuando el robot confirme que el componente está bien colocado. 
   // Para añadir un componente a una Mesa, simplemente se hace un OR con el contenido de la mesa y el material.
   // Una vez colocado el material en la mesa, se comprueba si ya están todos los materiales en esa caja para cerrarla y mandarla a la empaquetadora.
   IF "Estado5" THEN
       "SISTEMA_vbes".Mesa["SISTEMA_vbes".Mesa_EnProceso] := "SISTEMA_vbes".Mesa["SISTEMA_vbes".Mesa_EnProceso] OR "SISTEMA_vbes".Material_EnProceso;
       "SISTEMA_vbes".SP_Enmascarados := "SISTEMA_vbes".NumeroMateriales + 1;
       "SISTEMA_vbes".SP_Enmascarados := SHL(IN := 1, N := "SISTEMA_vbes".SP_Enmascarados);
       "SISTEMA_vbes".SP_Enmascarados := "SISTEMA_vbes".SP_Enmascarados - 1;
   END_IF;
   IF "Estado5" AND ("SISTEMA_vbes".Mesa["SISTEMA_vbes".Mesa_EnProceso] <> "SISTEMA_vbes".SP_Enmascarados) THEN
       "Estado0" := TRUE;
   END_IF;
   #_w1 := "Estado5";
   IF "Estado5" AND ("SISTEMA_vbes".Mesa["SISTEMA_vbes".Mesa_EnProceso] <> "SISTEMA_vbes".SP_Enmascarados) THEN
       "Estado5" := FALSE;
   END_IF;
   IF #_w1 AND ("SISTEMA_vbes".Mesa["SISTEMA_vbes".Mesa_EnProceso] = "SISTEMA_vbes".SP_Enmascarados) THEN
       "Estado6" := TRUE;
       "Estado5" := FALSE;
   END_IF;
   IF #_w1 THEN "SISTEMA_vbes".RobotOcupado := TRUE; END_IF;
END_REGION

REGION Network 8: Colocar tapadera
   // Cuando todos los componentes están colocados, se manda a poner una tapadera.
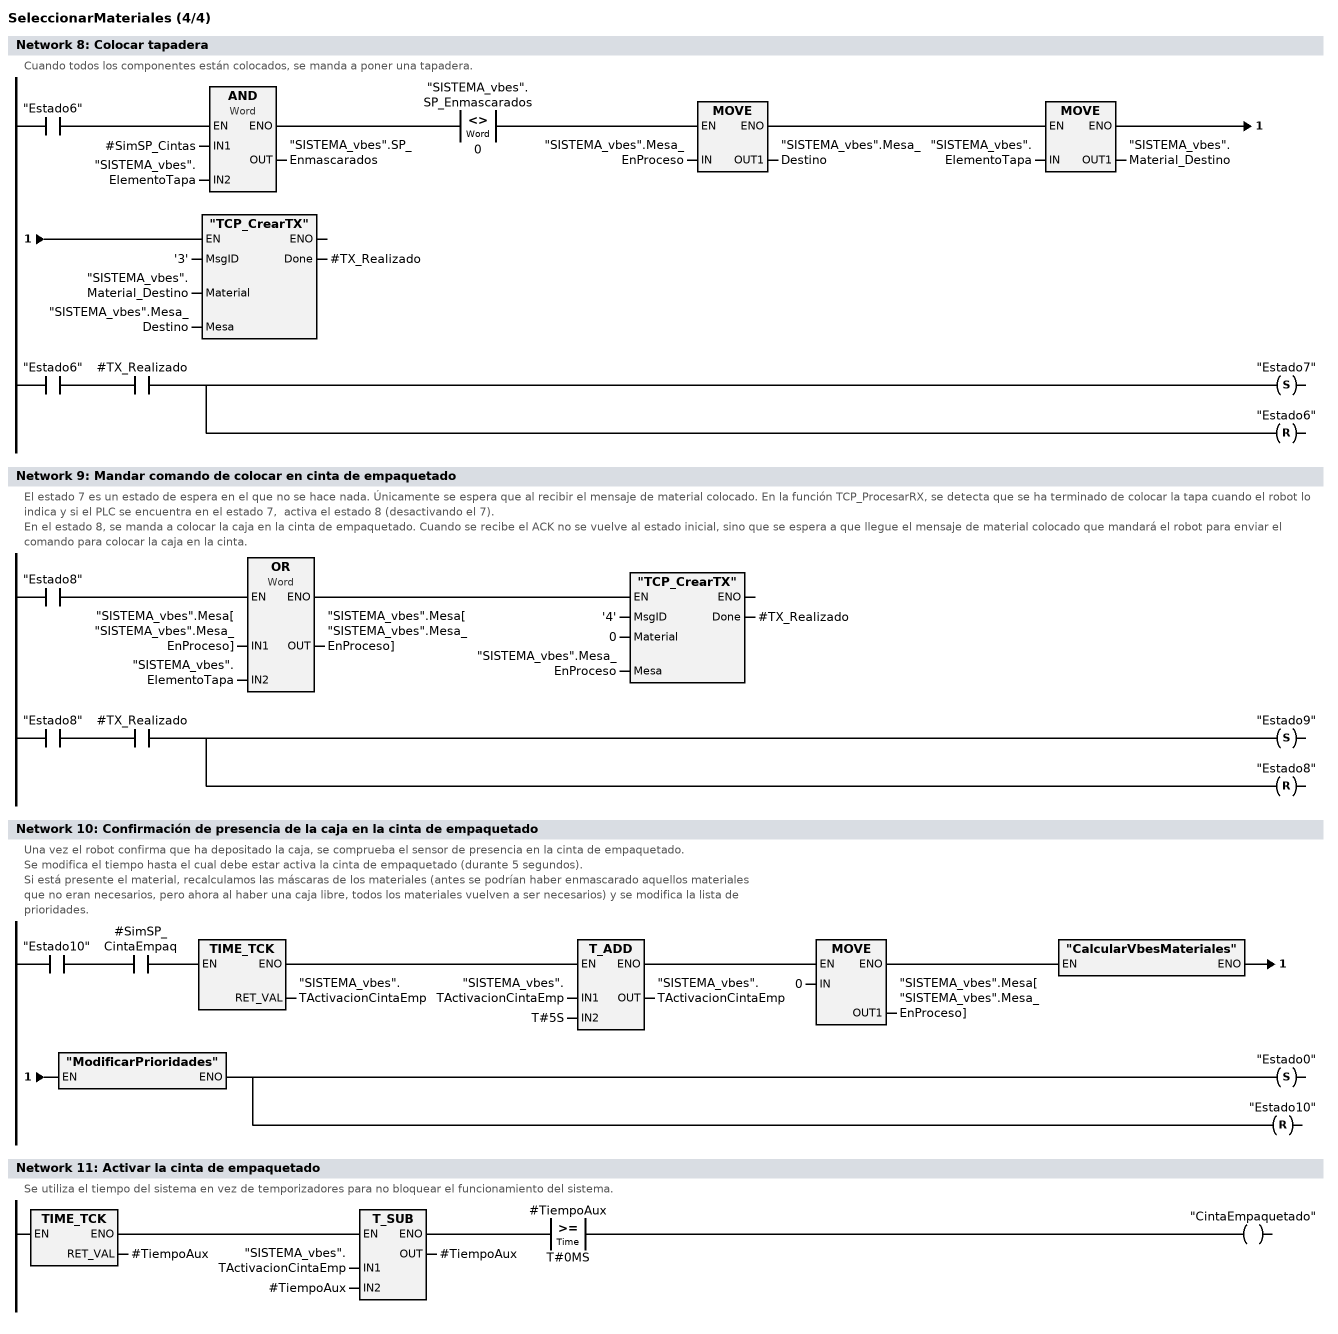
   RUNG wire#powerrail
      Contact( "Estado6" )
      { S7_Templates := "SrcType := Word" } And(in1 := #SimSP_Cintas, in2 := "SISTEMA_vbes".ElementoTapa, out => "SISTEMA_vbes".SP_Enmascarados)
      { S7_Templates := "SrcType := Word" } NE_Contact(in1 := "SISTEMA_vbes".SP_Enmascarados, in2 := 0)
      Move(in := "SISTEMA_vbes".Mesa_EnProceso, out1 => "SISTEMA_vbes".Mesa_Destino)
      Move(in := "SISTEMA_vbes".ElementoTapa, out1 => "SISTEMA_vbes".Material_Destino)
      "TCP_CrearTX"(MsgID := '3', Material := "SISTEMA_vbes".Material_Destino, Mesa := "SISTEMA_vbes".Mesa_Destino, Done => #TX_Realizado)
   END_RUNG
   RUNG wire#powerrail
      Contact( "Estado6" )
      Contact( #TX_Realizado )
      wire#w1
      S_Coil( "Estado7" )
   END_RUNG
   RUNG wire#w1
      R_Coil( "Estado6" )
   END_RUNG
   // the same network as SCL:
   IF "Estado6" THEN "SISTEMA_vbes".SP_Enmascarados := #SimSP_Cintas AND "SISTEMA_vbes".ElementoTapa; END_IF;
   IF "Estado6" AND ("SISTEMA_vbes".SP_Enmascarados <> 0) THEN
       "SISTEMA_vbes".Mesa_Destino := "SISTEMA_vbes".Mesa_EnProceso;
       "SISTEMA_vbes".Material_Destino := "SISTEMA_vbes".ElementoTapa;
       "TCP_CrearTX"(MsgID := '3',
                     Material := "SISTEMA_vbes".Material_Destino,
                     Mesa := "SISTEMA_vbes".Mesa_Destino,
                     Done => #TX_Realizado);
   END_IF;
   IF "Estado6" AND #TX_Realizado THEN
       "Estado7" := TRUE;
       "Estado6" := FALSE;
   END_IF;
END_REGION

REGION Network 9: Mandar comando de colocar en cinta de empaquetado
   // El estado 7 es un estado de espera en el que no se hace nada. Únicamente se espera que al recibir el mensaje de material colocado. En la función TCP_ProcesarRX, se detecta que se ha terminado de colocar la tapa cuando el robot lo indica y si el PLC se encuentra en el estado 7,  activa el estado 8 (desactivando el 7).
   // En el estado 8, se manda a colocar la caja en la cinta de empaquetado. Cuando se recibe el ACK no se vuelve al estado inicial, sino que se espera a que llegue el mensaje de material colocado que mandará el robot para enviar el comando para colocar la caja en la cinta.
   IF "Estado8" THEN
       "SISTEMA_vbes".Mesa["SISTEMA_vbes".Mesa_EnProceso] := "SISTEMA_vbes".Mesa["SISTEMA_vbes".Mesa_EnProceso] OR "SISTEMA_vbes".ElementoTapa;
       "TCP_CrearTX"(MsgID := '4', Material := 0, Mesa := "SISTEMA_vbes".Mesa_EnProceso, Done => #TX_Realizado);
   END_IF;
   IF "Estado8" AND #TX_Realizado THEN
       "Estado9" := TRUE;
       "Estado8" := FALSE;
   END_IF;
END_REGION

REGION Network 10: Confirmación de presencia de la caja en la cinta de empaquetado
   // Una vez el robot confirma que ha depositado la caja, se comprueba el sensor de presencia en la cinta de empaquetado.
   // Se modifica el tiempo hasta el cual debe estar activa la cinta de empaquetado (durante 5 segundos).
   // Si está presente el material, recalculamos las máscaras de los materiales (antes se podrían haber enmascarado aquellos materiales
   // que no eran necesarios, pero ahora al haber una caja libre, todos los materiales vuelven a ser necesarios) y se modifica la lista de 
   // prioridades.
   // ENO of a box is taken as its EN; it also drops when the box reports an error
   #_w1 := "Estado10" AND #SimSP_CintaEmpaq;
   IF #_w1 THEN
       "SISTEMA_vbes".TActivacionCintaEmp := TIME_TCK();
       "SISTEMA_vbes".TActivacionCintaEmp := T_ADD(IN1 := "SISTEMA_vbes".TActivacionCintaEmp, IN2 := T#5S);
       "SISTEMA_vbes".Mesa["SISTEMA_vbes".Mesa_EnProceso] := 0;
   END_IF;
   "CalcularVbesMateriales"(EN := #_w1, ENO => #_w2);
   "ModificarPrioridades"(EN := #_w2, ENO => #_w3);
   IF #_w3 THEN
       "Estado0" := TRUE;
       "Estado10" := FALSE;
   END_IF;
END_REGION

REGION Network 11: Activar la cinta de empaquetado
   // Se utiliza el tiempo del sistema en vez de temporizadores para no bloquear el funcionamiento del sistema.
   // ENO of a box is taken as its EN; it also drops when the box reports an error
   #TiempoAux := TIME_TCK();
   #TiempoAux := T_SUB(IN1 := "SISTEMA_vbes".TActivacionCintaEmp, IN2 := #TiempoAux);
   "CintaEmpaquetado" := #TiempoAux >= T#0MS;
END_REGION
END_FUNCTION

FUNCTION "ModificarPrioridades" : Void   // FC2, LAD
TITLE = Modificar prioridades
{ S7_Optimized_Access := 'TRUE' }
VERSION : 0.1
// Esta función desplaza la lista de prioridades cuando una caja está completada. La mesa actual pasa al final de la lista.
   VAR_TEMP
      IndiceBucle : Int;
      Temp : Int;
      SiguienteIndice : Int;
      FinalBucle : Int;
   END_VAR
BEGIN

REGION Network 1: Inicialización de variables
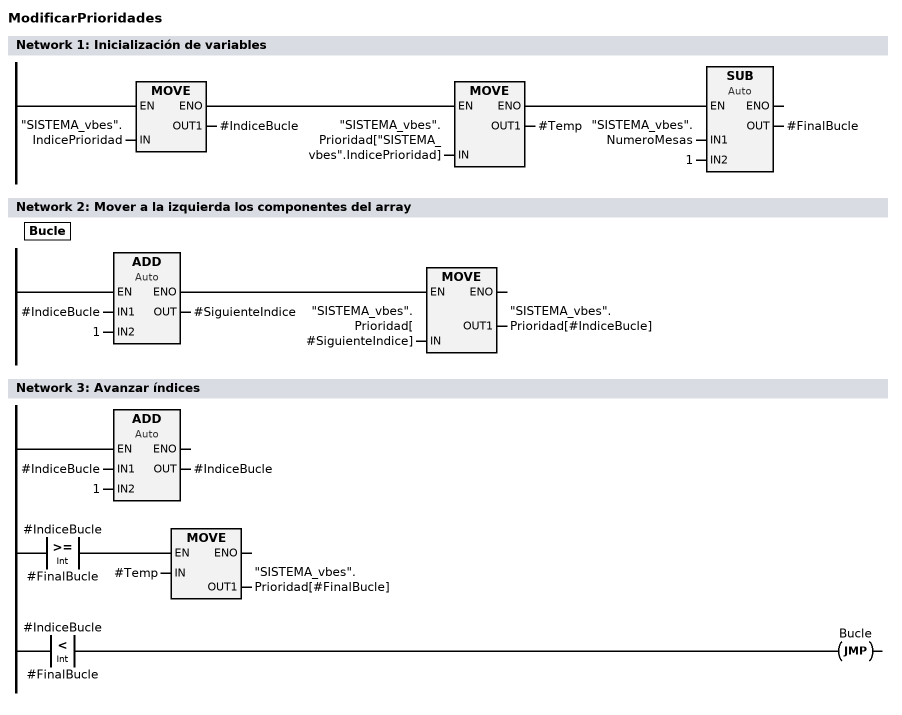
   RUNG wire#powerrail
      Move(in := "SISTEMA_vbes".IndicePrioridad, out1 => #IndiceBucle)
      Move(in := "SISTEMA_vbes".Prioridad["SISTEMA_vbes".IndicePrioridad], out1 => #Temp)
      Sub(in1 := "SISTEMA_vbes".NumeroMesas, in2 := 1, out => #FinalBucle)
   END_RUNG
   // the same network as SCL:
   #IndiceBucle := "SISTEMA_vbes".IndicePrioridad;
   #Temp := "SISTEMA_vbes".Prioridad["SISTEMA_vbes".IndicePrioridad];
   #FinalBucle := "SISTEMA_vbes".NumeroMesas - 1;
END_REGION

REGION Network 2: Mover a la izquierda los componentes del array
   Label( Bucle )
   RUNG wire#powerrail
      Add(in1 := #IndiceBucle, in2 := 1, out => #SiguienteIndice)
      Move(in := "SISTEMA_vbes".Prioridad[#SiguienteIndice], out1 => "SISTEMA_vbes".Prioridad[#IndiceBucle])
   END_RUNG
   // the same network as SCL:
   Bucle:
   #SiguienteIndice := #IndiceBucle + 1;
   "SISTEMA_vbes".Prioridad[#IndiceBucle] := "SISTEMA_vbes".Prioridad[#SiguienteIndice];
END_REGION

REGION Network 3: Avanzar índices
   RUNG wire#powerrail
      Add(in1 := #IndiceBucle, in2 := 1, out => #IndiceBucle)
   END_RUNG
   RUNG wire#powerrail
      { S7_Templates := "SrcType := Int" } GE_Contact(in1 := #IndiceBucle, in2 := #FinalBucle)
      Move(in := #Temp, out1 => "SISTEMA_vbes".Prioridad[#FinalBucle])
   END_RUNG
   RUNG wire#powerrail
      { S7_Templates := "SrcType := Int" } LT_Contact(in1 := #IndiceBucle, in2 := #FinalBucle)
      JumpCoil( Bucle )
   END_RUNG
   // the same network as SCL:
   #IndiceBucle := #IndiceBucle + 1;
   IF #IndiceBucle >= #FinalBucle THEN "SISTEMA_vbes".Prioridad[#FinalBucle] := #Temp; END_IF;
   IF #IndiceBucle < #FinalBucle THEN GOTO Bucle; END_IF;
END_REGION
END_FUNCTION

FUNCTION "TCP_CrearTX" : Void   // FC3, LAD
{ S7_Optimized_Access := 'TRUE' }
VERSION : 0.1
   VAR_INPUT
      MsgID : Char;
      Material : Word;
      Mesa : Int;
   END_VAR
   VAR_OUTPUT
      Done : Bool;
   END_VAR
   VAR_TEMP
      NoACK : Bool;   // Si el mensaje no necesita ACK marcar como TRUE
      TempCnt : UInt;
      ArgsStr : String;
      MesaByte : Byte;
      MsgListo : Bool;
   END_VAR
   VAR_TEMP   // added for the SCL form of the ladder/FBD networks
      _w1 : Bool;
   END_VAR
BEGIN

REGION Network 1: Si ya se está procesando un mensaje, el bloque no continuará su ejecución
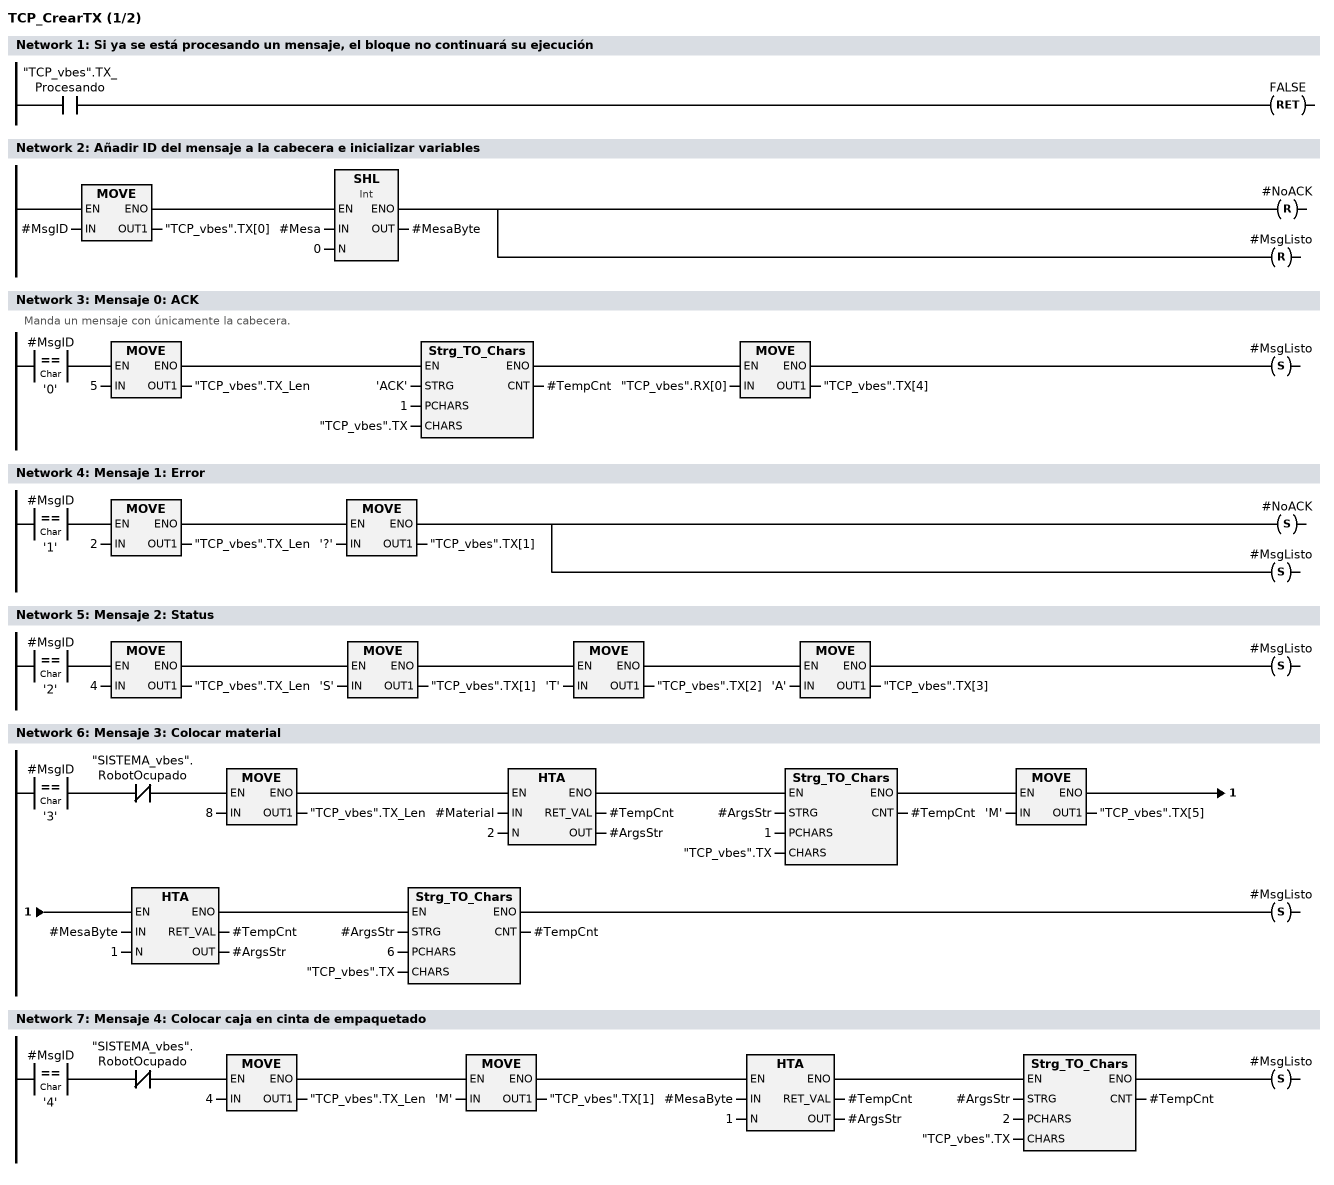
   IF "TCP_vbes".TX_Procesando THEN
       ENO := FALSE;
       RETURN;
   END_IF;
END_REGION

REGION Network 2: Añadir ID del mensaje a la cabecera e inicializar variables
   RUNG wire#powerrail
      Move(in := #MsgID, out1 => "TCP_vbes".TX[0])
      { S7_Templates := "SrcType := Int" } Shl(in := #Mesa, n := 0, out => #MesaByte)
      wire#w1
      R_Coil( #NoACK )
   END_RUNG
   RUNG wire#w1
      R_Coil( #MsgListo )
   END_RUNG
   // the same network as SCL:
   "TCP_vbes".TX[0] := #MsgID;
   #MesaByte := SHL(IN := #Mesa, N := 0);
   #NoACK := FALSE;
   #MsgListo := FALSE;
END_REGION

REGION Network 3: Mensaje 0: ACK
   // Manda un mensaje con únicamente la cabecera.
   // no SCL statement known for Strg_TO_Chars: written as a call
   // ENO of a box is taken as its EN; it also drops when the box reports an error
   IF #MsgID = '0' THEN
       "TCP_vbes".TX_Len := 5;
       Strg_TO_Chars(Strg := 'ACK', pChars := 1, Chars := "TCP_vbes".TX, Cnt => #TempCnt);
       "TCP_vbes".TX[4] := "TCP_vbes".RX[0];
       #MsgListo := TRUE;
   END_IF;
END_REGION

REGION Network 4: Mensaje 1: Error
   RUNG wire#powerrail
      { S7_Templates := "SrcType := Char" } EQ_Contact(in1 := #MsgID, in2 := '1')
      Move(in := 2, out1 => "TCP_vbes".TX_Len)
      Move(in := '?', out1 => "TCP_vbes".TX[1])
      wire#w1
      S_Coil( #NoACK )
   END_RUNG
   RUNG wire#w1
      S_Coil( #MsgListo )
   END_RUNG
   // the same network as SCL:
   IF #MsgID = '1' THEN
       "TCP_vbes".TX_Len := 2;
       "TCP_vbes".TX[1] := '?';
       #NoACK := TRUE;
       #MsgListo := TRUE;
   END_IF;
END_REGION

REGION Network 5: Mensaje 2: Status
   RUNG wire#powerrail
      { S7_Templates := "SrcType := Char" } EQ_Contact(in1 := #MsgID, in2 := '2')
      Move(in := 4, out1 => "TCP_vbes".TX_Len)
      Move(in := 'S', out1 => "TCP_vbes".TX[1])
      Move(in := 'T', out1 => "TCP_vbes".TX[2])
      Move(in := 'A', out1 => "TCP_vbes".TX[3])
      S_Coil( #MsgListo )
   END_RUNG
   // the same network as SCL:
   IF #MsgID = '2' THEN
       "TCP_vbes".TX_Len := 4;
       "TCP_vbes".TX[1] := 'S';
       "TCP_vbes".TX[2] := 'T';
       "TCP_vbes".TX[3] := 'A';
       #MsgListo := TRUE;
   END_IF;
END_REGION

REGION Network 6: Mensaje 3: Colocar material
   // no SCL statement known for Strg_TO_Chars: written as a call
   // ENO of a box is taken as its EN; it also drops when the box reports an error
   IF (#MsgID = '3') AND NOT "SISTEMA_vbes".RobotOcupado THEN "TCP_vbes".TX_Len := 8; END_IF;
   #_w1 := (#MsgID = '3') AND NOT "SISTEMA_vbes".RobotOcupado;
   IF #_w1 THEN
       #TempCnt := HTA(IN := #Material, N := 2, OUT => #ArgsStr);
       Strg_TO_Chars(Strg := #ArgsStr, pChars := 1, Chars := "TCP_vbes".TX, Cnt => #TempCnt);
       "TCP_vbes".TX[5] := 'M';
       #TempCnt := HTA(IN := #MesaByte, N := 1, OUT => #ArgsStr);
       Strg_TO_Chars(Strg := #ArgsStr, pChars := 6, Chars := "TCP_vbes".TX, Cnt => #TempCnt);
       #MsgListo := TRUE;
   END_IF;
END_REGION

REGION Network 7: Mensaje 4: Colocar caja en cinta de empaquetado
   // no SCL statement known for Strg_TO_Chars: written as a call
   // ENO of a box is taken as its EN; it also drops when the box reports an error
   IF (#MsgID = '4') AND NOT "SISTEMA_vbes".RobotOcupado THEN
       "TCP_vbes".TX_Len := 4;
       "TCP_vbes".TX[1] := 'M';
   END_IF;
   #_w1 := (#MsgID = '4') AND NOT "SISTEMA_vbes".RobotOcupado;
   IF #_w1 THEN
       #TempCnt := HTA(IN := #MesaByte, N := 1, OUT => #ArgsStr);
       Strg_TO_Chars(Strg := #ArgsStr, pChars := 2, Chars := "TCP_vbes".TX, Cnt => #TempCnt);
       #MsgListo := TRUE;
   END_IF;
END_REGION

REGION Network 8: Mensaje 5: Mandar valores de configuración
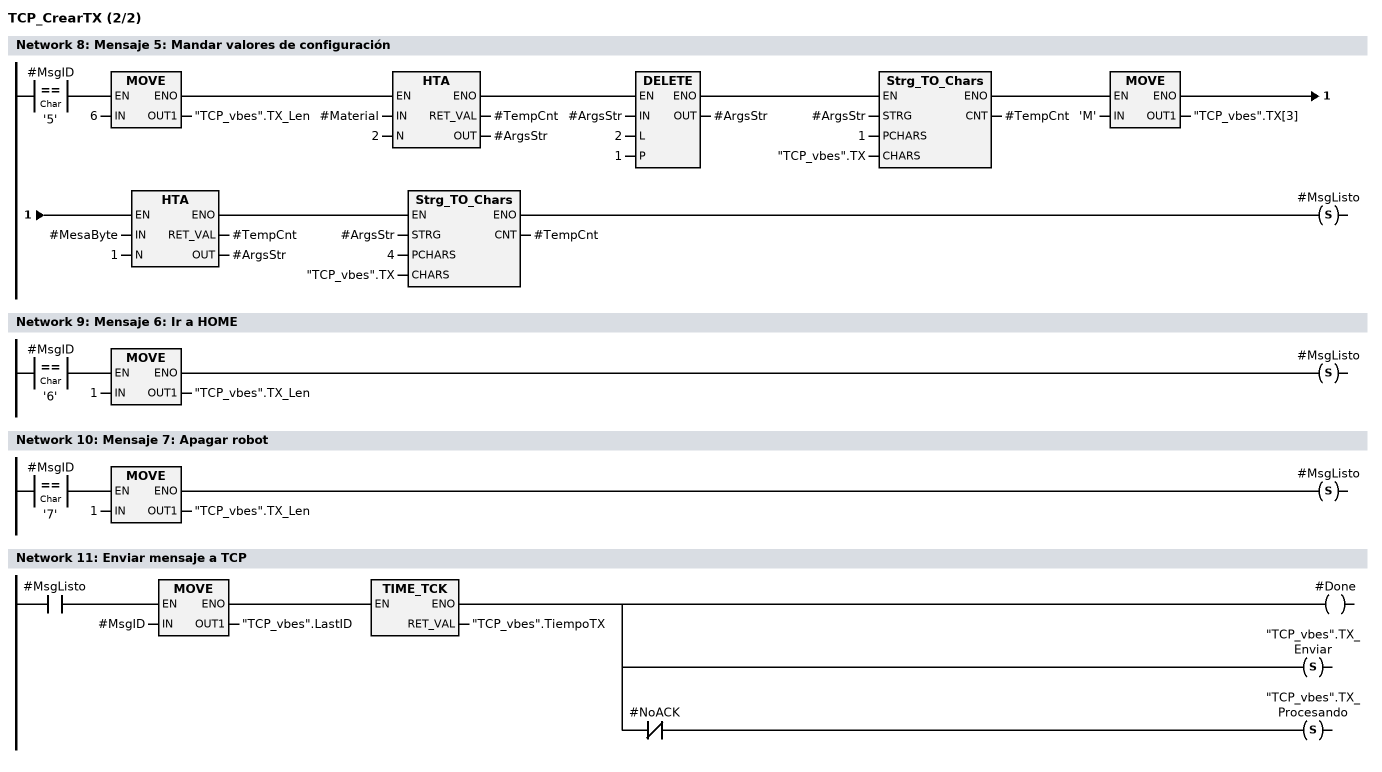
   // no SCL statement known for Strg_TO_Chars: written as a call
   // ENO of a box is taken as its EN; it also drops when the box reports an error
   IF #MsgID = '5' THEN
       "TCP_vbes".TX_Len := 6;
       #TempCnt := HTA(IN := #Material, N := 2, OUT => #ArgsStr);
       #ArgsStr := DELETE(IN := #ArgsStr, L := 2, P := 1);
       Strg_TO_Chars(Strg := #ArgsStr, pChars := 1, Chars := "TCP_vbes".TX, Cnt => #TempCnt);
       "TCP_vbes".TX[3] := 'M';
       #TempCnt := HTA(IN := #MesaByte, N := 1, OUT => #ArgsStr);
       Strg_TO_Chars(Strg := #ArgsStr, pChars := 4, Chars := "TCP_vbes".TX, Cnt => #TempCnt);
       #MsgListo := TRUE;
   END_IF;
END_REGION

REGION Network 9: Mensaje 6: Ir a HOME
   RUNG wire#powerrail
      { S7_Templates := "SrcType := Char" } EQ_Contact(in1 := #MsgID, in2 := '6')
      Move(in := 1, out1 => "TCP_vbes".TX_Len)
      S_Coil( #MsgListo )
   END_RUNG
   // the same network as SCL:
   IF #MsgID = '6' THEN
       "TCP_vbes".TX_Len := 1;
       #MsgListo := TRUE;
   END_IF;
END_REGION

REGION Network 10: Mensaje 7: Apagar robot
   RUNG wire#powerrail
      { S7_Templates := "SrcType := Char" } EQ_Contact(in1 := #MsgID, in2 := '7')
      Move(in := 1, out1 => "TCP_vbes".TX_Len)
      S_Coil( #MsgListo )
   END_RUNG
   // the same network as SCL:
   IF #MsgID = '7' THEN
       "TCP_vbes".TX_Len := 1;
       #MsgListo := TRUE;
   END_IF;
END_REGION

REGION Network 11: Enviar mensaje a TCP
   // ENO of a box is taken as its EN; it also drops when the box reports an error
   IF #MsgListo THEN
       "TCP_vbes".LastID := #MsgID;
       "TCP_vbes".TiempoTX := TIME_TCK();
   END_IF;
   #Done := #MsgListo;
   IF #MsgListo THEN "TCP_vbes".TX_Enviar := TRUE; END_IF;
   IF #MsgListo AND NOT #NoACK THEN "TCP_vbes".TX_Procesando := TRUE; END_IF;
END_REGION
END_FUNCTION

FUNCTION "TCP_ProcesarRX" : Void   // FC4, LAD
{ S7_Optimized_Access := 'TRUE' }
VERSION : 0.1
   VAR_TEMP
      MsgID : Char;
      MsgOK : Bool;
      TiempoAux : Time;
      LongStr : UDInt;
   END_VAR
   VAR_TEMP   // added for the SCL form of the ladder/FBD networks
      _w1 : Bool;
   END_VAR
BEGIN

REGION Network 1: Comprobar el tiempo del último TX para ver si el sistema se ha desconectado
   // Se espera que el sistema devuelva un ACK. Si pasan más de cinco segundos se tomará que el sistema está desconectado.
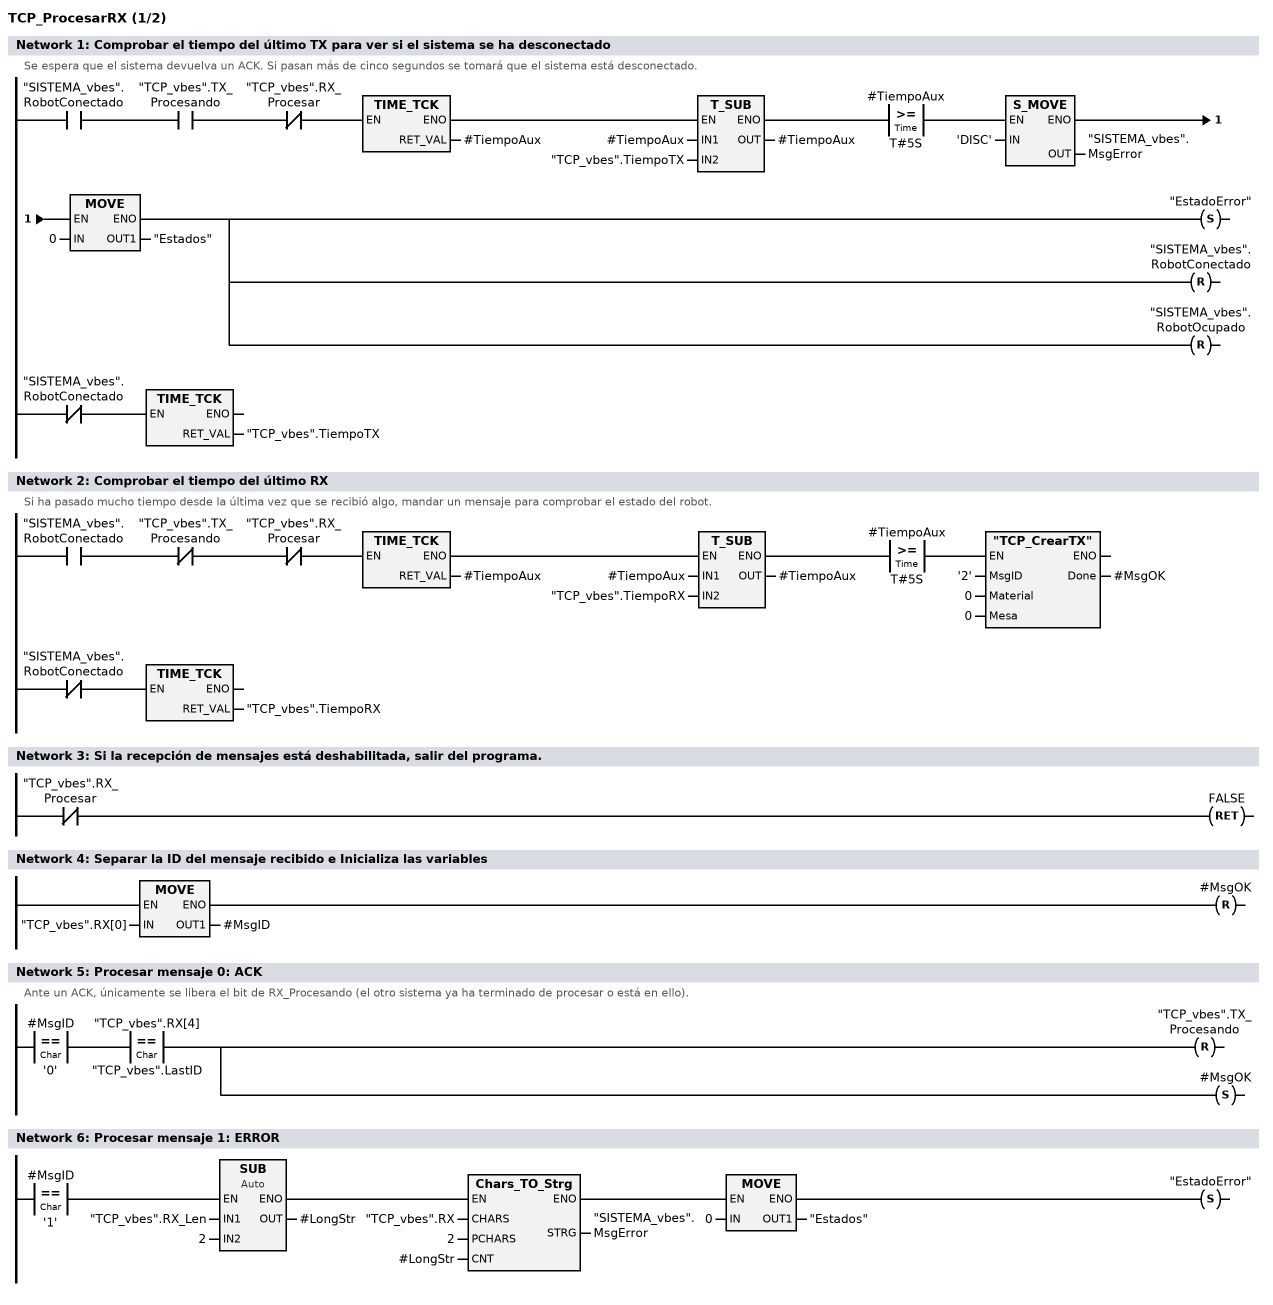
   // ENO of a box is taken as its EN; it also drops when the box reports an error
   #_w1 := "SISTEMA_vbes".RobotConectado AND "TCP_vbes".TX_Procesando AND NOT "TCP_vbes".RX_Procesar;
   IF #_w1 THEN
       #TiempoAux := TIME_TCK();
       #TiempoAux := T_SUB(IN1 := #TiempoAux, IN2 := "TCP_vbes".TiempoTX);
   END_IF;
   IF #_w1 AND (#TiempoAux >= T#5S) THEN
       "SISTEMA_vbes".MsgError := 'DISC';
       "Estados" := 0;
       "EstadoError" := TRUE;
       "SISTEMA_vbes".RobotConectado := FALSE;
       "SISTEMA_vbes".RobotOcupado := FALSE;
   END_IF;
   IF NOT "SISTEMA_vbes".RobotConectado THEN "TCP_vbes".TiempoTX := TIME_TCK(); END_IF;
END_REGION

REGION Network 2: Comprobar el tiempo del último RX
   // Si ha pasado mucho tiempo desde la última vez que se recibió algo, mandar un mensaje para comprobar el estado del robot.
   // ENO of a box is taken as its EN; it also drops when the box reports an error
   #_w1 := "SISTEMA_vbes".RobotConectado AND NOT "TCP_vbes".TX_Procesando AND NOT "TCP_vbes".RX_Procesar;
   IF #_w1 THEN
       #TiempoAux := TIME_TCK();
       #TiempoAux := T_SUB(IN1 := #TiempoAux, IN2 := "TCP_vbes".TiempoRX);
   END_IF;
   IF #_w1 AND (#TiempoAux >= T#5S) THEN
       "TCP_CrearTX"(MsgID := '2', Material := 0, Mesa := 0, Done => #MsgOK);
   END_IF;
   IF NOT "SISTEMA_vbes".RobotConectado THEN "TCP_vbes".TiempoRX := TIME_TCK(); END_IF;
END_REGION

REGION Network 3: Si la recepción de mensajes está deshabilitada, salir del programa.
   IF NOT "TCP_vbes".RX_Procesar THEN
       ENO := FALSE;
       RETURN;
   END_IF;
END_REGION

REGION Network 4: Separar la ID del mensaje recibido e Inicializa las variables
   RUNG wire#powerrail
      Move(in := "TCP_vbes".RX[0], out1 => #MsgID)
      R_Coil( #MsgOK )
   END_RUNG
   // the same network as SCL:
   #MsgID := "TCP_vbes".RX[0];
   #MsgOK := FALSE;
END_REGION

REGION Network 5: Procesar mensaje 0: ACK
   // Ante un ACK, únicamente se libera el bit de RX_Procesando (el otro sistema ya ha terminado de procesar o está en ello).
   RUNG wire#powerrail
      { S7_Templates := "SrcType := Char" } EQ_Contact(in1 := #MsgID, in2 := '0')
      { S7_Templates := "SrcType := Char" } EQ_Contact(in1 := "TCP_vbes".RX[4], in2 := "TCP_vbes".LastID)
      wire#w1
      R_Coil( "TCP_vbes".TX_Procesando )
   END_RUNG
   RUNG wire#w1
      S_Coil( #MsgOK )
   END_RUNG
   // the same network as SCL:
   IF (#MsgID = '0') AND ("TCP_vbes".RX[4] = "TCP_vbes".LastID) THEN
       "TCP_vbes".TX_Procesando := FALSE;
       #MsgOK := TRUE;
   END_IF;
END_REGION

REGION Network 6: Procesar mensaje 1: ERROR
   // no SCL statement known for Chars_TO_Strg: written as a call
   // ENO of a box is taken as its EN; it also drops when the box reports an error
   IF #MsgID = '1' THEN
       #LongStr := "TCP_vbes".RX_Len - 2;
       Chars_TO_Strg(Chars := "TCP_vbes".RX, pChars := 2, Cnt := #LongStr, Strg => "SISTEMA_vbes".MsgError);
       "Estados" := 0;
       "EstadoError" := TRUE;
   END_IF;
END_REGION

REGION Network 7: Procesar mensaje 2: Material recogido
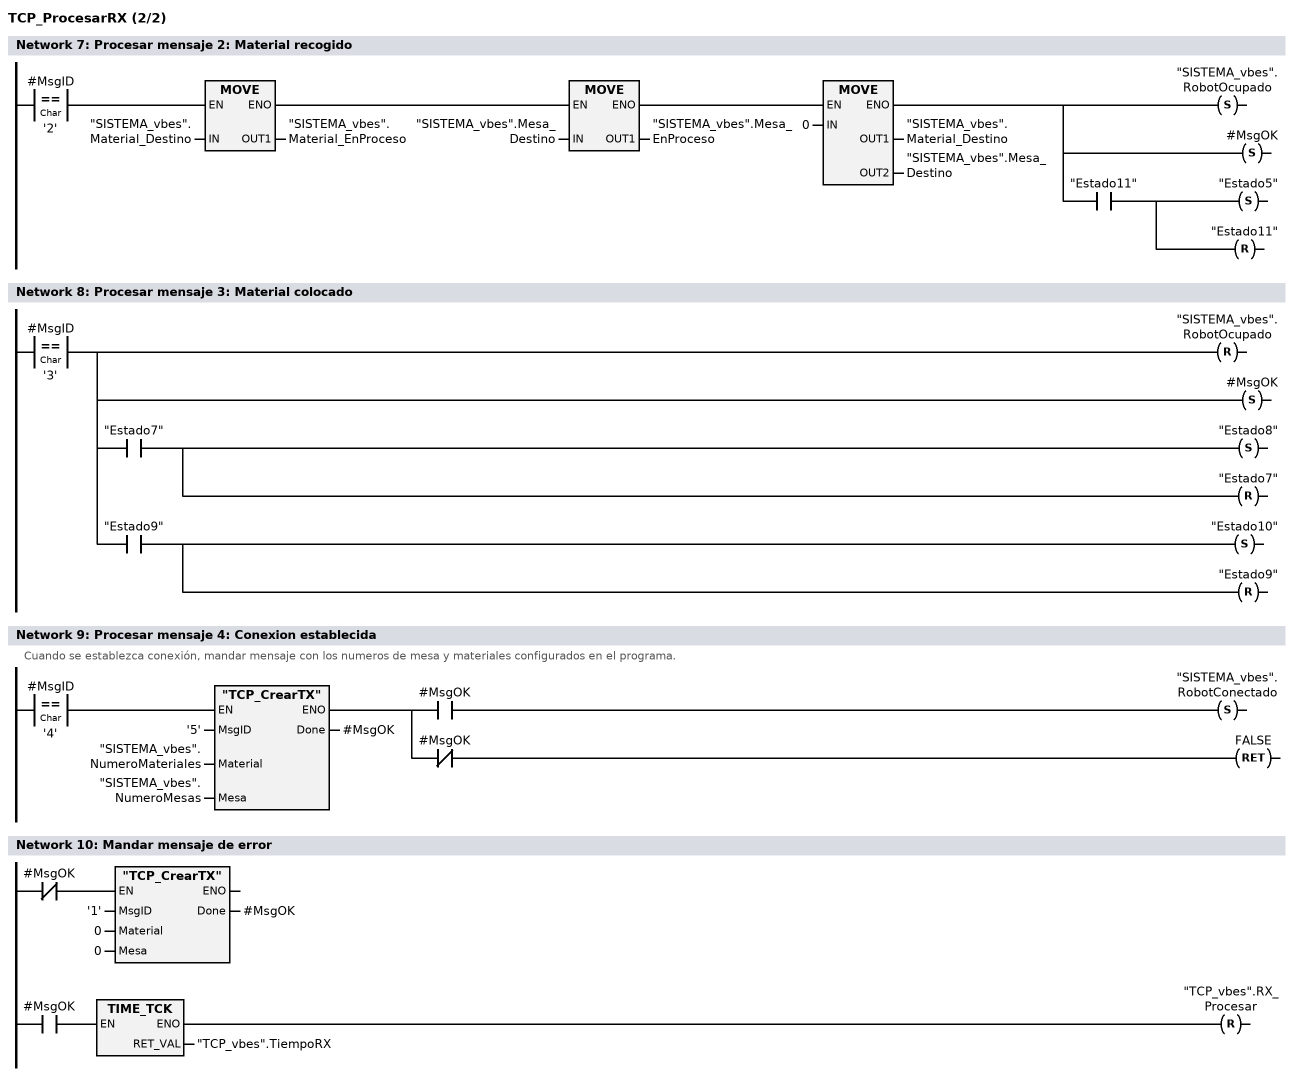
   RUNG wire#powerrail
      { S7_Templates := "SrcType := Char" } EQ_Contact(in1 := #MsgID, in2 := '2')
      Move(in := "SISTEMA_vbes".Material_Destino, out1 => "SISTEMA_vbes".Material_EnProceso)
      Move(in := "SISTEMA_vbes".Mesa_Destino, out1 => "SISTEMA_vbes".Mesa_EnProceso)
      Move(in := 0, out1 => "SISTEMA_vbes".Material_Destino, out2 => "SISTEMA_vbes".Mesa_Destino)
      wire#w1
      S_Coil( "SISTEMA_vbes".RobotOcupado )
   END_RUNG
   RUNG wire#w1
      S_Coil( #MsgOK )
   END_RUNG
   RUNG wire#w1
      Contact( "Estado11" )
      wire#w2
      S_Coil( "Estado5" )
   END_RUNG
   RUNG wire#w2
      R_Coil( "Estado11" )
   END_RUNG
   // the same network as SCL:
   #_w1 := #MsgID = '2';
   IF #_w1 THEN
       "SISTEMA_vbes".Material_EnProceso := "SISTEMA_vbes".Material_Destino;
       "SISTEMA_vbes".Mesa_EnProceso := "SISTEMA_vbes".Mesa_Destino;
       "SISTEMA_vbes".Material_Destino := 0;
       "SISTEMA_vbes".Mesa_Destino := 0;
       "SISTEMA_vbes".RobotOcupado := TRUE;
       #MsgOK := TRUE;
   END_IF;
   IF #_w1 AND "Estado11" THEN
       "Estado5" := TRUE;
       "Estado11" := FALSE;
   END_IF;
END_REGION

REGION Network 8: Procesar mensaje 3: Material colocado
   RUNG wire#powerrail
      { S7_Templates := "SrcType := Char" } EQ_Contact(in1 := #MsgID, in2 := '3')
      wire#w1
      R_Coil( "SISTEMA_vbes".RobotOcupado )
   END_RUNG
   RUNG wire#w1
      S_Coil( #MsgOK )
   END_RUNG
   RUNG wire#w1
      Contact( "Estado7" )
      wire#w2
      S_Coil( "Estado8" )
   END_RUNG
   RUNG wire#w2
      R_Coil( "Estado7" )
   END_RUNG
   RUNG wire#w1
      Contact( "Estado9" )
      wire#w3
      S_Coil( "Estado10" )
   END_RUNG
   RUNG wire#w3
      R_Coil( "Estado9" )
   END_RUNG
   // the same network as SCL:
   #_w1 := #MsgID = '3';
   IF #_w1 THEN
       "SISTEMA_vbes".RobotOcupado := FALSE;
       #MsgOK := TRUE;
   END_IF;
   IF #_w1 AND "Estado7" THEN
       "Estado8" := TRUE;
       "Estado7" := FALSE;
   END_IF;
   IF #_w1 AND "Estado9" THEN
       "Estado10" := TRUE;
       "Estado9" := FALSE;
   END_IF;
END_REGION

REGION Network 9: Procesar mensaje 4: Conexion establecida
   // Cuando se establezca conexión, mandar mensaje con los numeros de mesa y materiales configurados en el programa.
   "TCP_CrearTX"(EN := #MsgID = '4',
                 MsgID := '5',
                 Material := "SISTEMA_vbes".NumeroMateriales,
                 Mesa := "SISTEMA_vbes".NumeroMesas,
                 Done => #MsgOK,
                 ENO => #_w1);
   IF #_w1 AND #MsgOK THEN "SISTEMA_vbes".RobotConectado := TRUE; END_IF;
   IF #_w1 AND NOT #MsgOK THEN
       ENO := FALSE;
       RETURN;
   END_IF;
END_REGION

REGION Network 10: Mandar mensaje de error
   // ENO of a box is taken as its EN; it also drops when the box reports an error
   IF NOT #MsgOK THEN "TCP_CrearTX"(MsgID := '1', Material := 0, Mesa := 0, Done => #MsgOK); END_IF;
   IF #MsgOK THEN
       "TCP_vbes".TiempoRX := TIME_TCK();
       "TCP_vbes".RX_Procesar := FALSE;
   END_IF;
END_REGION
END_FUNCTION

FUNCTION "CalcularVbesMateriales" : Void   // FC5, LAD
TITLE = Calcular máscara de entrada y variables identificadoras según número de materiales
{ S7_Optimized_Access := 'TRUE' }
VERSION : 0.1
// Esta función sirve para crear las máscaras de entrada de los sensores de presencia de las cintas individuales. Los genera según el número de materiales que se haya especificado.
BEGIN

REGION Network 1: Cálculo de la máscara de COMPONENTES (excluyen base y tapa)
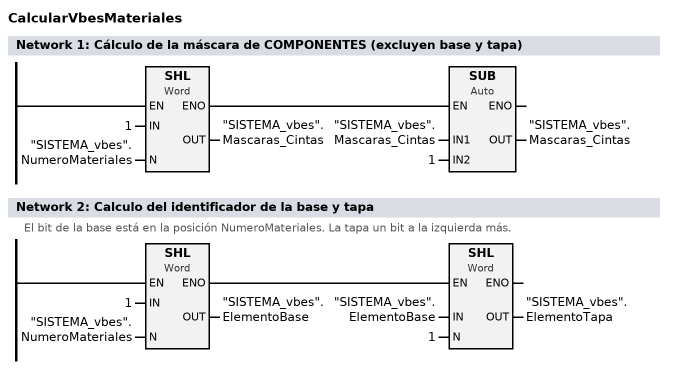
   RUNG wire#powerrail
      { S7_Templates := "SrcType := Word" } Shl(in := 1, n := "SISTEMA_vbes".NumeroMateriales, out => "SISTEMA_vbes".Mascaras_Cintas)
      Sub(in1 := "SISTEMA_vbes".Mascaras_Cintas, in2 := 1, out => "SISTEMA_vbes".Mascaras_Cintas)
   END_RUNG
   // the same network as SCL:
   "SISTEMA_vbes".Mascaras_Cintas := SHL(IN := 1, N := "SISTEMA_vbes".NumeroMateriales);
   "SISTEMA_vbes".Mascaras_Cintas := "SISTEMA_vbes".Mascaras_Cintas - 1;
END_REGION

REGION Network 2: Calculo del identificador de la base y tapa
   // El bit de la base está en la posición NumeroMateriales. La tapa un bit a la izquierda más.
   RUNG wire#powerrail
      { S7_Templates := "SrcType := Word" } Shl(in := 1, n := "SISTEMA_vbes".NumeroMateriales, out => "SISTEMA_vbes".ElementoBase)
      { S7_Templates := "SrcType := Word" } Shl(in := "SISTEMA_vbes".ElementoBase, n := 1, out => "SISTEMA_vbes".ElementoTapa)
   END_RUNG
   // the same network as SCL:
   "SISTEMA_vbes".ElementoBase := SHL(IN := 1, N := "SISTEMA_vbes".NumeroMateriales);
   "SISTEMA_vbes".ElementoTapa := SHL(IN := "SISTEMA_vbes".ElementoBase, N := 1);
END_REGION
END_FUNCTION

FUNCTION "GestionarErrores" : Void   // FC6, LAD
TITLE = Gestionar errores
{ S7_Optimized_Access := 'TRUE' }
VERSION : 0.1
   VAR_TEMP
      TempBool : Bool;
   END_VAR
BEGIN

REGION Network 1: Si no se encuentra en el estado de error, ignorar
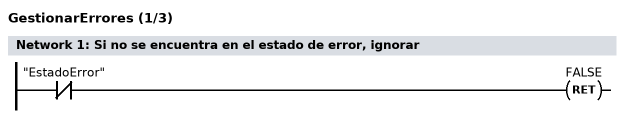
   IF NOT "EstadoError" THEN
       ENO := FALSE;
       RETURN;
   END_IF;
END_REGION

REGION Network 2: Crear bits para alarmas de estado en HMI
   // Se compara el string almacenado en MsgError con los mensajes conocidos y si es el mismo, se añade a los bits de errores.
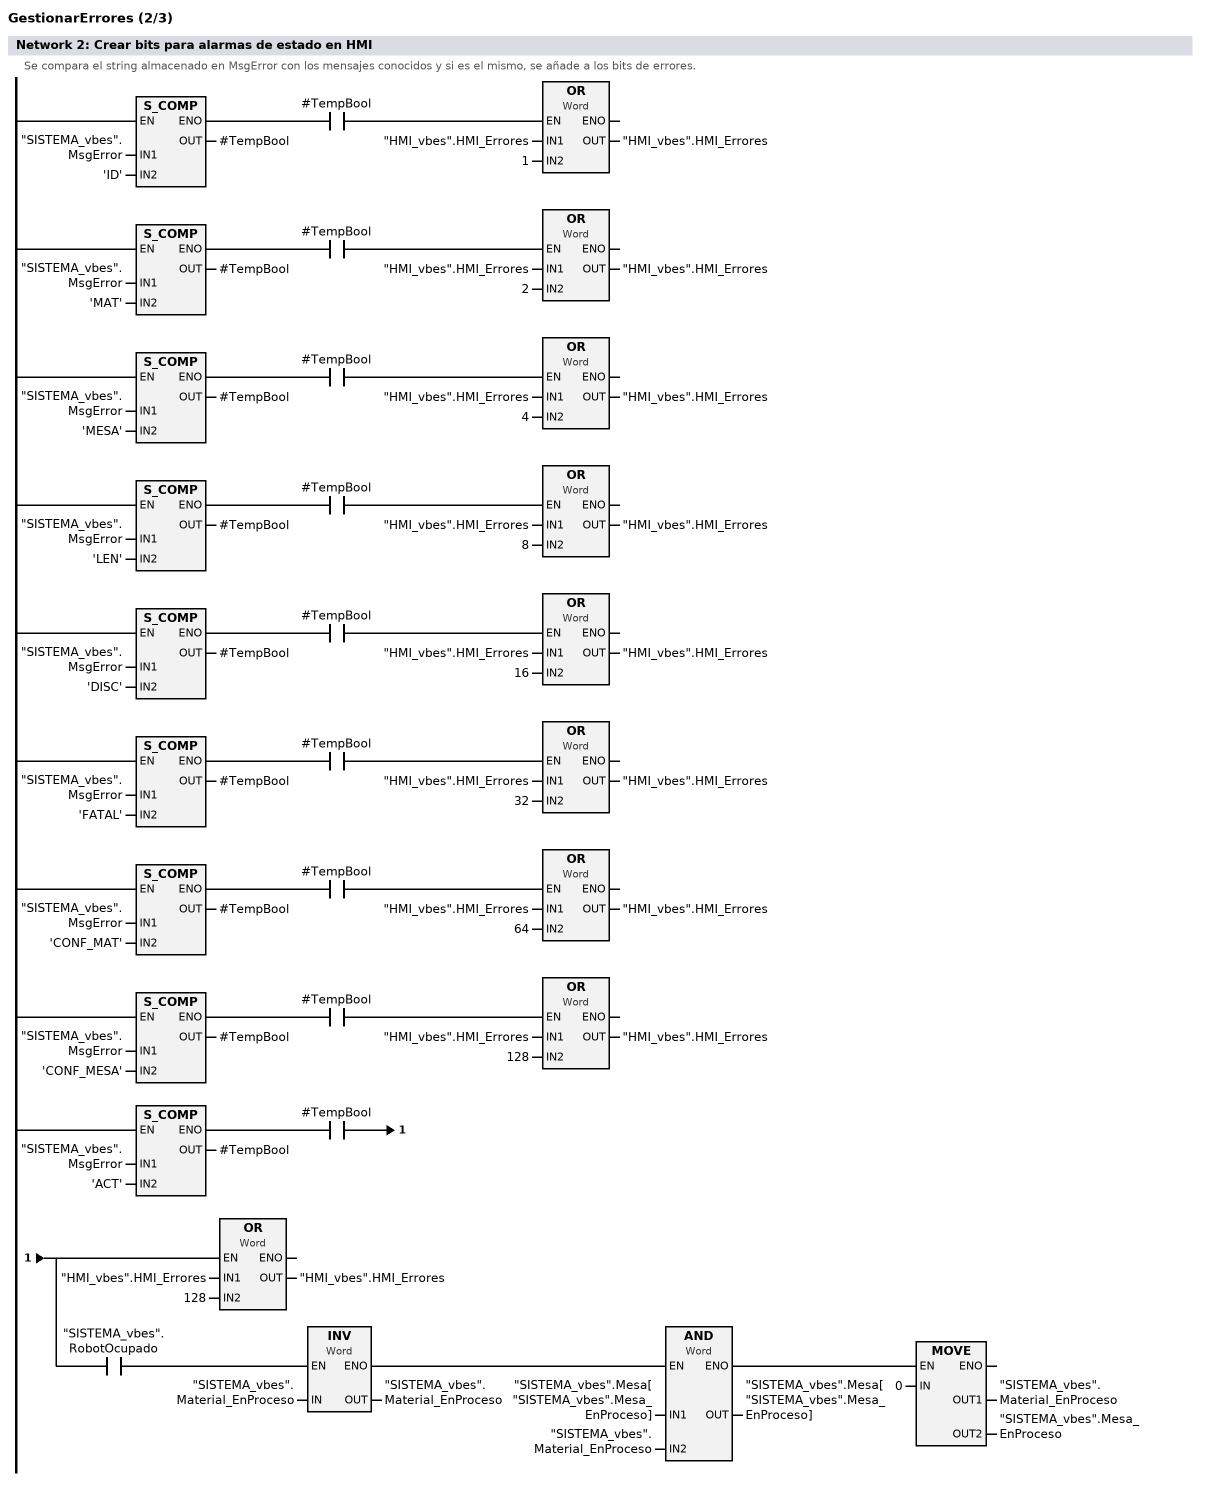
   // ENO of a box is taken as its EN; it also drops when the box reports an error
   S_COMP(IN1 := "SISTEMA_vbes".MsgError, IN2 := 'ID', OUT => #TempBool);
   IF #TempBool THEN "HMI_vbes".HMI_Errores := "HMI_vbes".HMI_Errores OR 1; END_IF;
   S_COMP(IN1 := "SISTEMA_vbes".MsgError, IN2 := 'MAT', OUT => #TempBool);
   IF #TempBool THEN "HMI_vbes".HMI_Errores := "HMI_vbes".HMI_Errores OR 2; END_IF;
   S_COMP(IN1 := "SISTEMA_vbes".MsgError, IN2 := 'MESA', OUT => #TempBool);
   IF #TempBool THEN "HMI_vbes".HMI_Errores := "HMI_vbes".HMI_Errores OR 4; END_IF;
   S_COMP(IN1 := "SISTEMA_vbes".MsgError, IN2 := 'LEN', OUT => #TempBool);
   IF #TempBool THEN "HMI_vbes".HMI_Errores := "HMI_vbes".HMI_Errores OR 8; END_IF;
   S_COMP(IN1 := "SISTEMA_vbes".MsgError, IN2 := 'DISC', OUT => #TempBool);
   IF #TempBool THEN "HMI_vbes".HMI_Errores := "HMI_vbes".HMI_Errores OR 16; END_IF;
   S_COMP(IN1 := "SISTEMA_vbes".MsgError, IN2 := 'FATAL', OUT => #TempBool);
   IF #TempBool THEN "HMI_vbes".HMI_Errores := "HMI_vbes".HMI_Errores OR 32; END_IF;
   S_COMP(IN1 := "SISTEMA_vbes".MsgError, IN2 := 'CONF_MAT', OUT => #TempBool);
   IF #TempBool THEN "HMI_vbes".HMI_Errores := "HMI_vbes".HMI_Errores OR 64; END_IF;
   S_COMP(IN1 := "SISTEMA_vbes".MsgError, IN2 := 'CONF_MESA', OUT => #TempBool);
   IF #TempBool THEN "HMI_vbes".HMI_Errores := "HMI_vbes".HMI_Errores OR 128; END_IF;
   S_COMP(IN1 := "SISTEMA_vbes".MsgError, IN2 := 'ACT', OUT => #TempBool);
   IF #TempBool THEN "HMI_vbes".HMI_Errores := "HMI_vbes".HMI_Errores OR 128; END_IF;
   IF #TempBool AND "SISTEMA_vbes".RobotOcupado THEN
       "SISTEMA_vbes".Material_EnProceso := NOT "SISTEMA_vbes".Material_EnProceso;
       "SISTEMA_vbes".Mesa["SISTEMA_vbes".Mesa_EnProceso] := "SISTEMA_vbes".Mesa["SISTEMA_vbes".Mesa_EnProceso] AND "SISTEMA_vbes".Material_EnProceso;
       "SISTEMA_vbes".Material_EnProceso := 0;
       "SISTEMA_vbes".Mesa_EnProceso := 0;
   END_IF;
END_REGION

REGION Network 3: Reiniciar errores y estados
   // En todos los casos, ante error el usuario debe reiniciar el sistema, aunque estaría mejor dicho rearmarlo.
   // Cuando el sistema es rearmado se vuelve al estado inicial pero se siguen almacenando los valores dentro de SISTEMA_vbes, luego el sistema continúa por dónde se quedó antes del error.
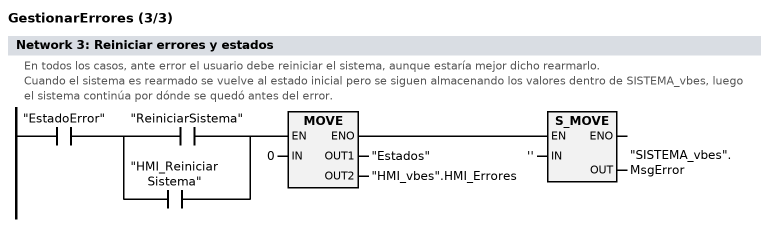
   RUNG wire#powerrail
      Contact( "EstadoError" )
      wire#w1
      Contact( "ReiniciarSistema" )
      wire#w2
      Move(in := 0, out1 => "Estados", out2 => "HMI_vbes".HMI_Errores)
      S_Move(in := '', out => "SISTEMA_vbes".MsgError)
   END_RUNG
   RUNG wire#w1
      Contact( "HMI_ReiniciarSistema" )
   END_RUNG wire#w2
   // the same network as SCL:
   IF "EstadoError" AND ("ReiniciarSistema" OR "HMI_ReiniciarSistema") THEN
       "Estados" := 0;
       "HMI_vbes".HMI_Errores := 0;
       "SISTEMA_vbes".MsgError := '';
   END_IF;
END_REGION
END_FUNCTION

FUNCTION "CalcularHMI" : Void   // FC7, LAD
{ S7_Optimized_Access := 'TRUE' }
VERSION : 0.1
   VAR_TEMP
      TempWord : Word;
      MandarConfRobot : Bool;   // True si ha habido un cambio y se debe mandar conf
   END_VAR
   VAR_TEMP   // added for the SCL form of the ladder/FBD networks
      _w1 : Bool;
   END_VAR
BEGIN

REGION Network 1: Generar los bools para que se muestren los componentes por mesa
   // En la primera rama se seleccionan únicamente los materiales (para el caso en el que el número de materiales de la bandeja es menor), para ello, se enmascaran.
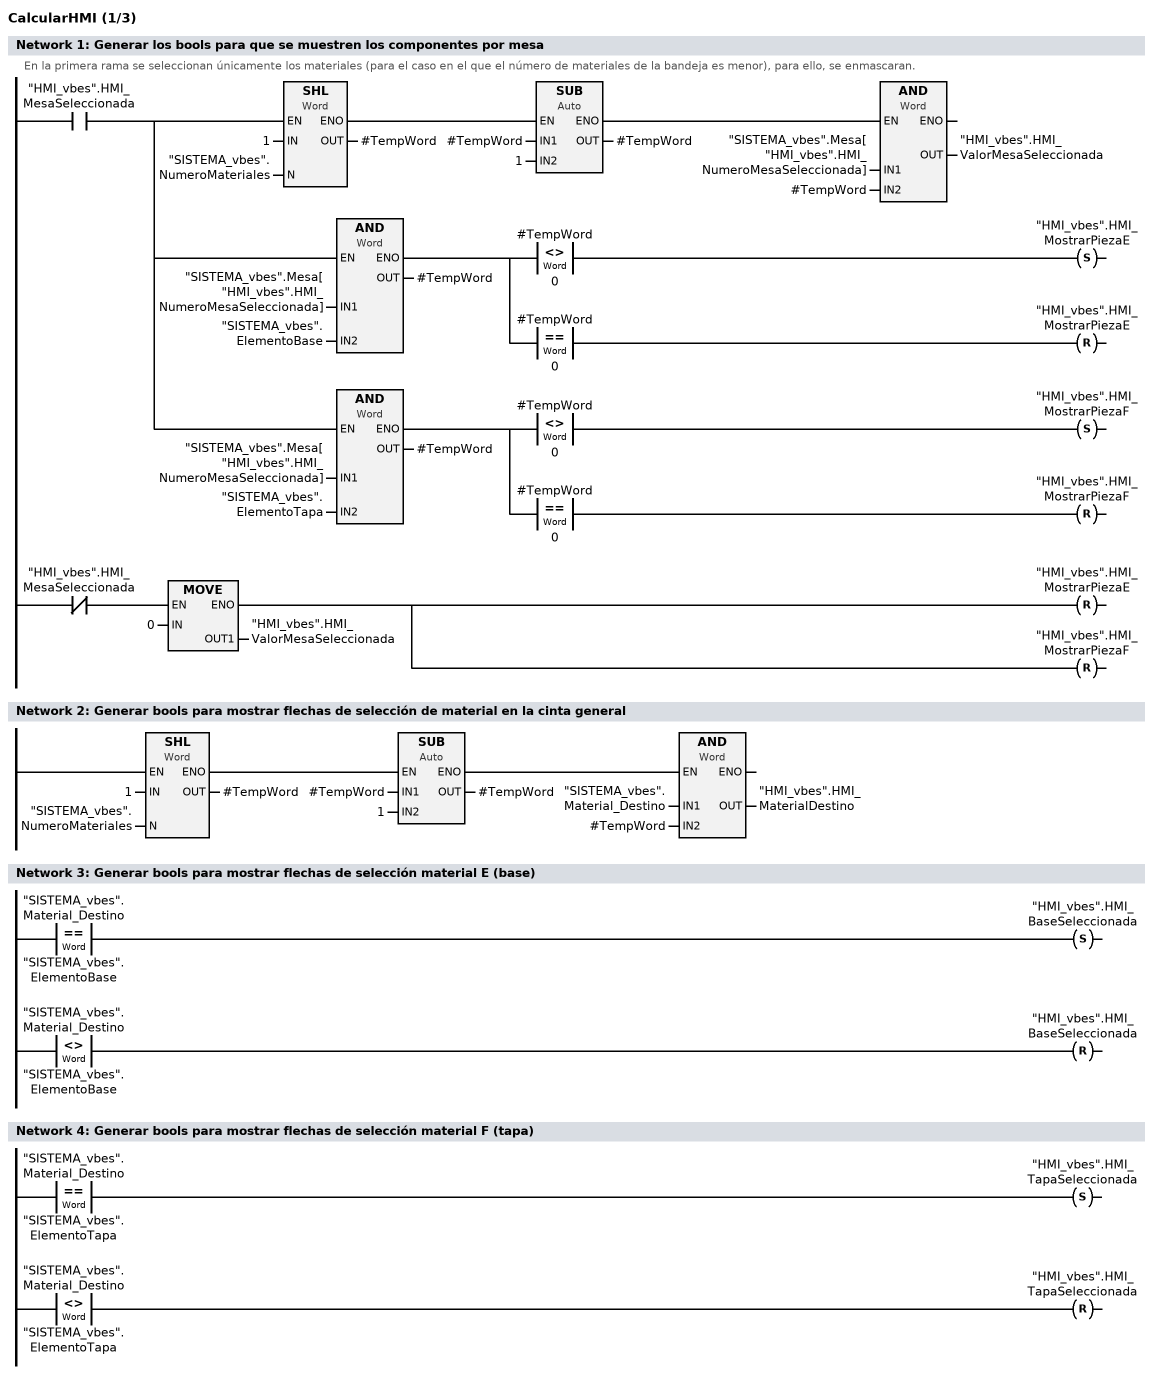
   RUNG wire#powerrail
      Contact( "HMI_vbes".HMI_MesaSeleccionada )
      wire#w1
      { S7_Templates := "SrcType := Word" } Shl(in := 1, n := "SISTEMA_vbes".NumeroMateriales, out => #TempWord)
      Sub(in1 := #TempWord, in2 := 1, out => #TempWord)
      { S7_Templates := "SrcType := Word" } And(in1 := "SISTEMA_vbes".Mesa["HMI_vbes".HMI_NumeroMesaSeleccionada], in2 := #TempWord, out => "HMI_vbes".HMI_ValorMesaSeleccionada)
   END_RUNG
   RUNG wire#w1
      { S7_Templates := "SrcType := Word" } And(in1 := "SISTEMA_vbes".Mesa["HMI_vbes".HMI_NumeroMesaSeleccionada], in2 := "SISTEMA_vbes".ElementoBase, out => #TempWord)
      wire#w2
      { S7_Templates := "SrcType := Word" } NE_Contact(in1 := #TempWord, in2 := 0)
      S_Coil( "HMI_vbes".HMI_MostrarPiezaE )
   END_RUNG
   RUNG wire#w2
      { S7_Templates := "SrcType := Word" } EQ_Contact(in1 := #TempWord, in2 := 0)
      R_Coil( "HMI_vbes".HMI_MostrarPiezaE )
   END_RUNG
   RUNG wire#w1
      { S7_Templates := "SrcType := Word" } And(in1 := "SISTEMA_vbes".Mesa["HMI_vbes".HMI_NumeroMesaSeleccionada], in2 := "SISTEMA_vbes".ElementoTapa, out => #TempWord)
      wire#w3
      { S7_Templates := "SrcType := Word" } NE_Contact(in1 := #TempWord, in2 := 0)
      S_Coil( "HMI_vbes".HMI_MostrarPiezaF )
   END_RUNG
   RUNG wire#w3
      { S7_Templates := "SrcType := Word" } EQ_Contact(in1 := #TempWord, in2 := 0)
      R_Coil( "HMI_vbes".HMI_MostrarPiezaF )
   END_RUNG
   RUNG wire#powerrail
      I_Contact( "HMI_vbes".HMI_MesaSeleccionada )
      Move(in := 0, out1 => "HMI_vbes".HMI_ValorMesaSeleccionada)
      wire#w4
      R_Coil( "HMI_vbes".HMI_MostrarPiezaE )
   END_RUNG
   RUNG wire#w4
      R_Coil( "HMI_vbes".HMI_MostrarPiezaF )
   END_RUNG
   // the same network as SCL:
   IF "HMI_vbes".HMI_MesaSeleccionada THEN
       #TempWord := SHL(IN := 1, N := "SISTEMA_vbes".NumeroMateriales);
       #TempWord := #TempWord - 1;
       "HMI_vbes".HMI_ValorMesaSeleccionada := "SISTEMA_vbes".Mesa["HMI_vbes".HMI_NumeroMesaSeleccionada] AND #TempWord;
       #TempWord := "SISTEMA_vbes".Mesa["HMI_vbes".HMI_NumeroMesaSeleccionada] AND "SISTEMA_vbes".ElementoBase;
   END_IF;
   IF "HMI_vbes".HMI_MesaSeleccionada AND (#TempWord <> 0) THEN "HMI_vbes".HMI_MostrarPiezaE := TRUE; END_IF;
   IF "HMI_vbes".HMI_MesaSeleccionada AND (#TempWord = 0) THEN "HMI_vbes".HMI_MostrarPiezaE := FALSE; END_IF;
   IF "HMI_vbes".HMI_MesaSeleccionada THEN
       #TempWord := "SISTEMA_vbes".Mesa["HMI_vbes".HMI_NumeroMesaSeleccionada] AND "SISTEMA_vbes".ElementoTapa;
   END_IF;
   IF "HMI_vbes".HMI_MesaSeleccionada AND (#TempWord <> 0) THEN "HMI_vbes".HMI_MostrarPiezaF := TRUE; END_IF;
   IF "HMI_vbes".HMI_MesaSeleccionada AND (#TempWord = 0) THEN "HMI_vbes".HMI_MostrarPiezaF := FALSE; END_IF;
   IF NOT "HMI_vbes".HMI_MesaSeleccionada THEN
       "HMI_vbes".HMI_ValorMesaSeleccionada := 0;
       "HMI_vbes".HMI_MostrarPiezaE := FALSE;
       "HMI_vbes".HMI_MostrarPiezaF := FALSE;
   END_IF;
END_REGION

REGION Network 2: Generar bools para mostrar flechas de selección de material en la cinta general
   RUNG wire#powerrail
      { S7_Templates := "SrcType := Word" } Shl(in := 1, n := "SISTEMA_vbes".NumeroMateriales, out => #TempWord)
      Sub(in1 := #TempWord, in2 := 1, out => #TempWord)
      { S7_Templates := "SrcType := Word" } And(in1 := "SISTEMA_vbes".Material_Destino, in2 := #TempWord, out => "HMI_vbes".HMI_MaterialDestino)
   END_RUNG
   // the same network as SCL:
   #TempWord := SHL(IN := 1, N := "SISTEMA_vbes".NumeroMateriales);
   #TempWord := #TempWord - 1;
   "HMI_vbes".HMI_MaterialDestino := "SISTEMA_vbes".Material_Destino AND #TempWord;
END_REGION

REGION Network 3: Generar bools para mostrar flechas de selección material E (base)
   RUNG wire#powerrail
      { S7_Templates := "SrcType := Word" } EQ_Contact(in1 := "SISTEMA_vbes".Material_Destino, in2 := "SISTEMA_vbes".ElementoBase)
      S_Coil( "HMI_vbes".HMI_BaseSeleccionada )
   END_RUNG
   RUNG wire#powerrail
      { S7_Templates := "SrcType := Word" } NE_Contact(in1 := "SISTEMA_vbes".Material_Destino, in2 := "SISTEMA_vbes".ElementoBase)
      R_Coil( "HMI_vbes".HMI_BaseSeleccionada )
   END_RUNG
   // the same network as SCL:
   IF "SISTEMA_vbes".Material_Destino = "SISTEMA_vbes".ElementoBase THEN
       "HMI_vbes".HMI_BaseSeleccionada := TRUE;
   END_IF;
   IF "SISTEMA_vbes".Material_Destino <> "SISTEMA_vbes".ElementoBase THEN
       "HMI_vbes".HMI_BaseSeleccionada := FALSE;
   END_IF;
END_REGION

REGION Network 4: Generar bools para mostrar flechas de selección material F (tapa)
   RUNG wire#powerrail
      { S7_Templates := "SrcType := Word" } EQ_Contact(in1 := "SISTEMA_vbes".Material_Destino, in2 := "SISTEMA_vbes".ElementoTapa)
      S_Coil( "HMI_vbes".HMI_TapaSeleccionada )
   END_RUNG
   RUNG wire#powerrail
      { S7_Templates := "SrcType := Word" } NE_Contact(in1 := "SISTEMA_vbes".Material_Destino, in2 := "SISTEMA_vbes".ElementoTapa)
      R_Coil( "HMI_vbes".HMI_TapaSeleccionada )
   END_RUNG
   // the same network as SCL:
   IF "SISTEMA_vbes".Material_Destino = "SISTEMA_vbes".ElementoTapa THEN
       "HMI_vbes".HMI_TapaSeleccionada := TRUE;
   END_IF;
   IF "SISTEMA_vbes".Material_Destino <> "SISTEMA_vbes".ElementoTapa THEN
       "HMI_vbes".HMI_TapaSeleccionada := FALSE;
   END_IF;
END_REGION

REGION Network 5: Mostrar colores de la mesa seleccionada
   // Se coloca un número grande para que no se seleccione ningún botón (esto es porque las mesas empiezan desde el número cero, luego ese valor neutral encendería el botón de la mesa cero). Si el sistema se encuentra en alguno de los estados donde tiene una mesa seleccionada, se pasa el valor real de la mesa al HMI.
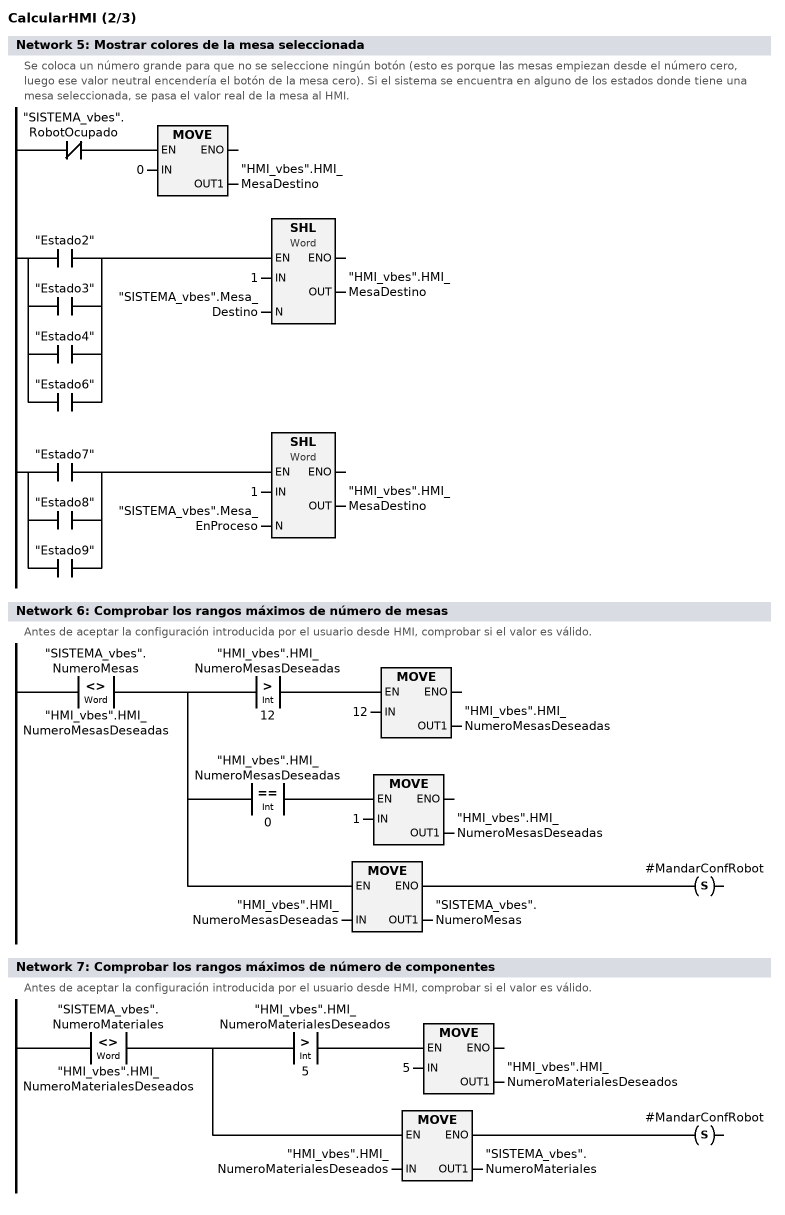
   RUNG wire#powerrail
      I_Contact( "SISTEMA_vbes".RobotOcupado )
      Move(in := 0, out1 => "HMI_vbes".HMI_MesaDestino)
   END_RUNG
   RUNG wire#powerrail
      Contact( "Estado2" )
      wire#w1
      { S7_Templates := "SrcType := Word" } Shl(in := 1, n := "SISTEMA_vbes".Mesa_Destino, out => "HMI_vbes".HMI_MesaDestino)
   END_RUNG
   RUNG wire#powerrail
      Contact( "Estado3" )
   END_RUNG wire#w1
   RUNG wire#powerrail
      Contact( "Estado4" )
   END_RUNG wire#w1
   RUNG wire#powerrail
      Contact( "Estado6" )
   END_RUNG wire#w1
   RUNG wire#powerrail
      Contact( "Estado7" )
      wire#w2
      { S7_Templates := "SrcType := Word" } Shl(in := 1, n := "SISTEMA_vbes".Mesa_EnProceso, out => "HMI_vbes".HMI_MesaDestino)
   END_RUNG
   RUNG wire#powerrail
      Contact( "Estado8" )
   END_RUNG wire#w2
   RUNG wire#powerrail
      Contact( "Estado9" )
   END_RUNG wire#w2
   // the same network as SCL:
   IF NOT "SISTEMA_vbes".RobotOcupado THEN "HMI_vbes".HMI_MesaDestino := 0; END_IF;
   IF "Estado2" OR "Estado3" OR "Estado4" OR "Estado6" THEN
       "HMI_vbes".HMI_MesaDestino := SHL(IN := 1, N := "SISTEMA_vbes".Mesa_Destino);
   END_IF;
   IF "Estado7" OR "Estado8" OR "Estado9" THEN
       "HMI_vbes".HMI_MesaDestino := SHL(IN := 1, N := "SISTEMA_vbes".Mesa_EnProceso);
   END_IF;
END_REGION

REGION Network 6: Comprobar los rangos máximos de número de mesas
   // Antes de aceptar la configuración introducida por el usuario desde HMI, comprobar si el valor es válido.
   RUNG wire#powerrail
      { S7_Templates := "SrcType := Word" } NE_Contact(in1 := "SISTEMA_vbes".NumeroMesas, in2 := "HMI_vbes".HMI_NumeroMesasDeseadas)
      wire#w1
      { S7_Templates := "SrcType := Int" } GT_Contact(in1 := "HMI_vbes".HMI_NumeroMesasDeseadas, in2 := 12)
      Move(in := 12, out1 => "HMI_vbes".HMI_NumeroMesasDeseadas)
   END_RUNG
   RUNG wire#w1
      { S7_Templates := "SrcType := Int" } EQ_Contact(in1 := "HMI_vbes".HMI_NumeroMesasDeseadas, in2 := 0)
      Move(in := 1, out1 => "HMI_vbes".HMI_NumeroMesasDeseadas)
   END_RUNG
   RUNG wire#w1
      Move(in := "HMI_vbes".HMI_NumeroMesasDeseadas, out1 => "SISTEMA_vbes".NumeroMesas)
      S_Coil( #MandarConfRobot )
   END_RUNG
   // the same network as SCL:
   #_w1 := "SISTEMA_vbes".NumeroMesas <> "HMI_vbes".HMI_NumeroMesasDeseadas;
   IF #_w1 AND ("HMI_vbes".HMI_NumeroMesasDeseadas > 12) THEN
       "HMI_vbes".HMI_NumeroMesasDeseadas := 12;
   END_IF;
   IF #_w1 AND ("HMI_vbes".HMI_NumeroMesasDeseadas = 0) THEN "HMI_vbes".HMI_NumeroMesasDeseadas := 1; END_IF;
   IF #_w1 THEN
       "SISTEMA_vbes".NumeroMesas := "HMI_vbes".HMI_NumeroMesasDeseadas;
       #MandarConfRobot := TRUE;
   END_IF;
END_REGION

REGION Network 7: Comprobar los rangos máximos de número de componentes
   // Antes de aceptar la configuración introducida por el usuario desde HMI, comprobar si el valor es válido.
   RUNG wire#powerrail
      { S7_Templates := "SrcType := Word" } NE_Contact(in1 := "SISTEMA_vbes".NumeroMateriales, in2 := "HMI_vbes".HMI_NumeroMaterialesDeseados)
      wire#w1
      { S7_Templates := "SrcType := Int" } GT_Contact(in1 := "HMI_vbes".HMI_NumeroMaterialesDeseados, in2 := 5)
      Move(in := 5, out1 => "HMI_vbes".HMI_NumeroMaterialesDeseados)
   END_RUNG
   RUNG wire#w1
      Move(in := "HMI_vbes".HMI_NumeroMaterialesDeseados, out1 => "SISTEMA_vbes".NumeroMateriales)
      S_Coil( #MandarConfRobot )
   END_RUNG
   // the same network as SCL:
   #_w1 := "SISTEMA_vbes".NumeroMateriales <> "HMI_vbes".HMI_NumeroMaterialesDeseados;
   IF #_w1 AND ("HMI_vbes".HMI_NumeroMaterialesDeseados > 5) THEN
       "HMI_vbes".HMI_NumeroMaterialesDeseados := 5;
   END_IF;
   IF #_w1 THEN
       "SISTEMA_vbes".NumeroMateriales := "HMI_vbes".HMI_NumeroMaterialesDeseados;
       #MandarConfRobot := TRUE;
   END_IF;
END_REGION

REGION Network 8: Si hay configuración nueva, mandarla al robot
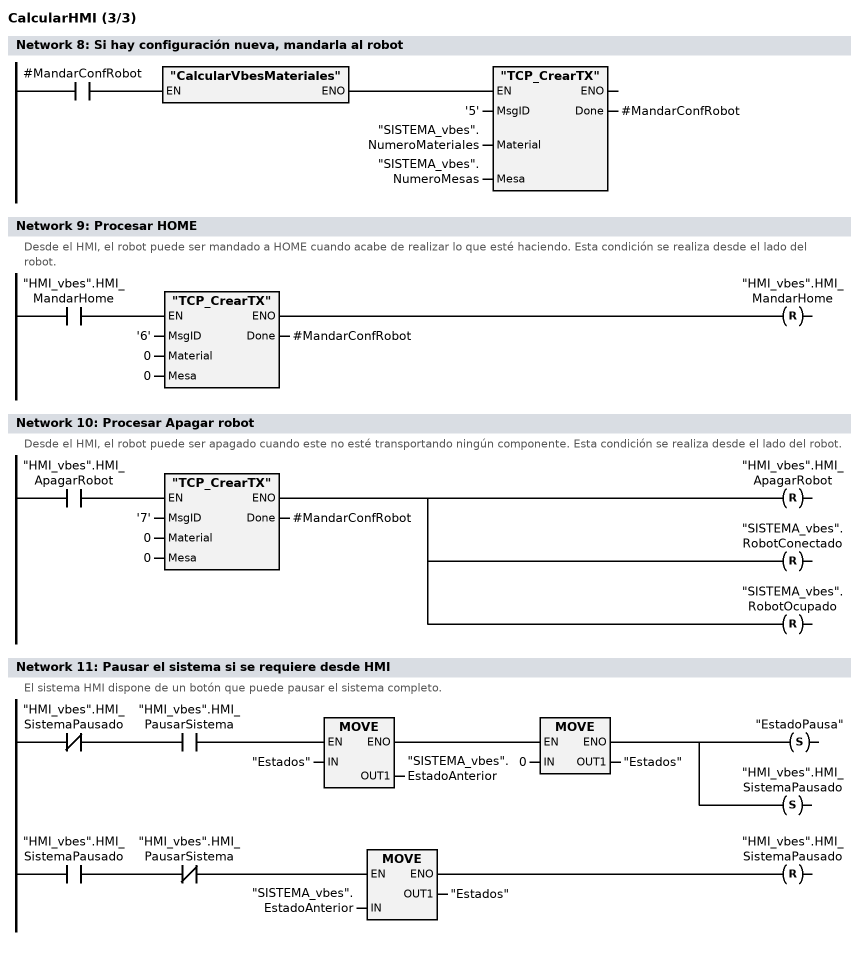
   RUNG wire#powerrail
      Contact( #MandarConfRobot )
      "CalcularVbesMateriales"()
      "TCP_CrearTX"(MsgID := '5', Material := "SISTEMA_vbes".NumeroMateriales, Mesa := "SISTEMA_vbes".NumeroMesas, Done => #MandarConfRobot)
   END_RUNG
   // the same network as SCL:
   "CalcularVbesMateriales"(EN := #MandarConfRobot, ENO => #_w1);
   IF #_w1 THEN
       "TCP_CrearTX"(MsgID := '5',
                     Material := "SISTEMA_vbes".NumeroMateriales,
                     Mesa := "SISTEMA_vbes".NumeroMesas,
                     Done => #MandarConfRobot);
   END_IF;
END_REGION

REGION Network 9: Procesar HOME
   // Desde el HMI, el robot puede ser mandado a HOME cuando acabe de realizar lo que esté haciendo. Esta condición se realiza desde el lado del robot.
   RUNG wire#powerrail
      Contact( "HMI_vbes".HMI_MandarHome )
      "TCP_CrearTX"(MsgID := '6', Material := 0, Mesa := 0, Done => #MandarConfRobot)
      R_Coil( "HMI_vbes".HMI_MandarHome )
   END_RUNG
   // the same network as SCL:
   "TCP_CrearTX"(EN := "HMI_vbes".HMI_MandarHome,
                 MsgID := '6',
                 Material := 0,
                 Mesa := 0,
                 Done => #MandarConfRobot,
                 ENO => #_w1);
   IF #_w1 THEN "HMI_vbes".HMI_MandarHome := FALSE; END_IF;
END_REGION

REGION Network 10: Procesar Apagar robot
   // Desde el HMI, el robot puede ser apagado cuando este no esté transportando ningún componente. Esta condición se realiza desde el lado del robot.
   RUNG wire#powerrail
      Contact( "HMI_vbes".HMI_ApagarRobot )
      "TCP_CrearTX"(MsgID := '7', Material := 0, Mesa := 0, Done => #MandarConfRobot)
      wire#w1
      R_Coil( "HMI_vbes".HMI_ApagarRobot )
   END_RUNG
   RUNG wire#w1
      R_Coil( "SISTEMA_vbes".RobotConectado )
   END_RUNG
   RUNG wire#w1
      R_Coil( "SISTEMA_vbes".RobotOcupado )
   END_RUNG
   // the same network as SCL:
   "TCP_CrearTX"(EN := "HMI_vbes".HMI_ApagarRobot,
                 MsgID := '7',
                 Material := 0,
                 Mesa := 0,
                 Done => #MandarConfRobot,
                 ENO => #_w1);
   IF #_w1 THEN
       "HMI_vbes".HMI_ApagarRobot := FALSE;
       "SISTEMA_vbes".RobotConectado := FALSE;
       "SISTEMA_vbes".RobotOcupado := FALSE;
   END_IF;
END_REGION

REGION Network 11: Pausar el sistema si se requiere desde HMI
   // El sistema HMI dispone de un botón que puede pausar el sistema completo.
   RUNG wire#powerrail
      I_Contact( "HMI_vbes".HMI_SistemaPausado )
      Contact( "HMI_vbes".HMI_PausarSistema )
      Move(in := "Estados", out1 => "SISTEMA_vbes".EstadoAnterior)
      Move(in := 0, out1 => "Estados")
      wire#w1
      S_Coil( "EstadoPausa" )
   END_RUNG
   RUNG wire#w1
      S_Coil( "HMI_vbes".HMI_SistemaPausado )
   END_RUNG
   RUNG wire#powerrail
      Contact( "HMI_vbes".HMI_SistemaPausado )
      I_Contact( "HMI_vbes".HMI_PausarSistema )
      Move(in := "SISTEMA_vbes".EstadoAnterior, out1 => "Estados")
      R_Coil( "HMI_vbes".HMI_SistemaPausado )
   END_RUNG
   // the same network as SCL:
   IF NOT "HMI_vbes".HMI_SistemaPausado AND "HMI_vbes".HMI_PausarSistema THEN
       "SISTEMA_vbes".EstadoAnterior := "Estados";
       "Estados" := 0;
       "EstadoPausa" := TRUE;
       "HMI_vbes".HMI_SistemaPausado := TRUE;
   END_IF;
   IF "HMI_vbes".HMI_SistemaPausado AND NOT "HMI_vbes".HMI_PausarSistema THEN
       "Estados" := "SISTEMA_vbes".EstadoAnterior;
       "HMI_vbes".HMI_SistemaPausado := FALSE;
   END_IF;
END_REGION
END_FUNCTION

ORGANIZATION_BLOCK "Main"   // OB1, LAD, ProgramCycle
TITLE = "Main Program Sweep (Cycle)"
{ S7_Optimized_Access := 'TRUE' }
VERSION : 0.1
   VAR_INPUT
      Initial_Call : Bool;   // Initial call of this OB
      Remanence : Bool;   // =True, if remanent data are available
   END_VAR
   VAR_TEMP
      DummyBool : Bool;
   END_VAR
   VAR_TEMP   // added for the SCL form of the ladder/FBD networks
      _w1 : Bool;
   END_VAR
BEGIN

REGION Network 1: Inicialización del sistema
   // Si el sistema acaba de arrancar (todos los estados están a 0), vuelve al estado inicial  0.
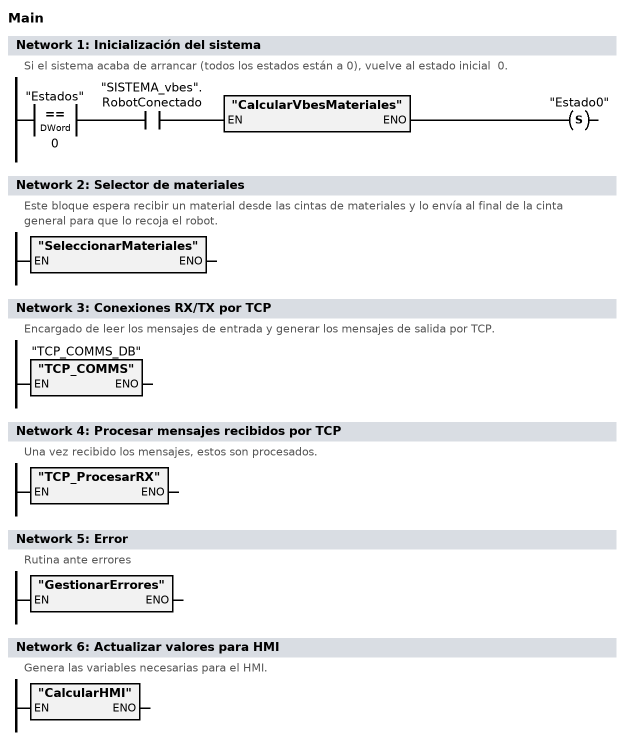
   RUNG wire#powerrail
      { S7_Templates := "SrcType := DWord" } EQ_Contact(in1 := "Estados", in2 := 0)
      Contact( "SISTEMA_vbes".RobotConectado )
      "CalcularVbesMateriales"()
      S_Coil( "Estado0" )
   END_RUNG
   // the same network as SCL:
   "CalcularVbesMateriales"(EN := ("Estados" = 0) AND "SISTEMA_vbes".RobotConectado, ENO => #_w1);
   IF #_w1 THEN "Estado0" := TRUE; END_IF;
END_REGION

REGION Network 2: Selector de materiales
   // Este bloque espera recibir un material desde las cintas de materiales y lo envía al final de la cinta general para que lo recoja el robot.
   RUNG wire#powerrail
      "SeleccionarMateriales"()
   END_RUNG
   // the same network as SCL:
   "SeleccionarMateriales"();
END_REGION

REGION Network 3: Conexiones RX/TX por TCP
   // Encargado de leer los mensajes de entrada y generar los mensajes de salida por TCP.
   RUNG wire#powerrail
      "TCP_COMMS_DB"()
   END_RUNG
   // the same network as SCL:
   "TCP_COMMS_DB"();   // "TCP_COMMS"
END_REGION

REGION Network 4: Procesar mensajes recibidos por TCP
   // Una vez recibido los mensajes, estos son procesados.
   RUNG wire#powerrail
      "TCP_ProcesarRX"()
   END_RUNG
   // the same network as SCL:
   "TCP_ProcesarRX"();
END_REGION

REGION Network 5: Error
   // Rutina ante errores
   RUNG wire#powerrail
      "GestionarErrores"()
   END_RUNG
   // the same network as SCL:
   "GestionarErrores"();
END_REGION

REGION Network 6: Actualizar valores para HMI
   // Genera las variables necesarias para el HMI.
   RUNG wire#powerrail
      "CalcularHMI"()
   END_RUNG
   // the same network as SCL:
   "CalcularHMI"();
END_REGION
END_ORGANIZATION_BLOCK

(* ===== HMI "HMI_RT_1" =====
system functions are stored by id; their names below are inferred from use
connection "HMI_Connection_1": ETHERNET, S7_1500_OMS

HMI tags "Default tag table"
   "Tag_ScreenNumber" : UInt, internal
   "vbes_RobotConectado" : Bool = PLC SISTEMA_vbes.RobotConectado AT %DB8.DBX86.1, 100 ms
   "SP_CintaGeneral" : Bool = PLC SP_CintaGeneral AT %E1.6, 100 ms
   "CintaGeneral" : Bool = PLC CintaGeneral AT %A1.6, 100 ms
   "vbes_RobotOcupado" : Bool = PLC SISTEMA_vbes.RobotOcupado AT %DB8.DBX86.0, 100 ms
   "CintaEmpaquetado" : Bool = PLC CintaEmpaquetado AT %A1.7, 100 ms
   "HMI_SP_Cintas" : Word = PLC HMI_SP_Cintas AT %MW10, 100 ms
   "SP_Cintas" : Word = PLC SP_Cintas AT %EW0, 100 ms
   "SP_CintaEmpaquetado" : Bool = PLC SP_CintaEmpaquetado AT %E1.7, 100 ms
   "vbes_Material_Destino" : Word = PLC SISTEMA_vbes.Material_Destino AT %DB8.DBW64, 100 ms
   "vbes_ModoSimulacion" : Bool = PLC SISTEMA_vbes.ModoSimulacion AT %DB8.DBX348.0, 100 ms
   "HMI_SP_CintaGeneral" : Bool = PLC HMI_SP_CintaGeneral AT %M11.6, 100 ms
   "HMI_SP_CintaEmpaquetado" : Bool = PLC HMI_SP_CintaEmpaquetado AT %M11.7, 100 ms
   "SP_CintaGeneral_Forzado" : Bool AT %DB1.DBX0.0
   "SP_CintaEmpaq_Forzado" : Bool AT %DB1.DBX0.0
   "MesaSeleccionada" : Bool = PLC HMI_vbes.HMI_MesaSeleccionada AT %DB9.DBX4.0, 100 ms
   "HMI_PaleE" : Bool = PLC HMI_PaleE AT %M12.0, 100 ms
   "HMI_PaleF" : Bool = PLC HMI_PaleF AT %M12.1, 100 ms
   "NumeroMesaSeleccionada" : Int = PLC HMI_vbes.HMI_NumeroMesaSeleccionada AT %DB9.DBW0, 100 ms
   "vbes_NumeroMesas" : Word = PLC SISTEMA_vbes.NumeroMesas AT %DB8.DBW74, 100 ms
   "vbes_ElementoBase" : Word = PLC SISTEMA_vbes.ElementoBase AT %DB8.DBW344, 100 ms
   "vbes_ElementoTapa" : Word = PLC SISTEMA_vbes.ElementoTapa AT %DB8.DBW346, 100 ms
   "HMI_TapaSeleccionada" : Bool = PLC HMI_vbes.HMI_TapaSeleccionada AT %DB9.DBX4.2, 100 ms
   "HMI_BaseSeleccionada" : Bool = PLC HMI_vbes.HMI_BaseSeleccionada AT %DB9.DBX4.1, 100 ms
   "vbes_NumeroMateriales" : Int = PLC SISTEMA_vbes.NumeroMateriales AT %DB8.DBW84, 100 ms
   "HMI_MesasDisponiblesDeseadas" : Int = PLC HMI_vbes.HMI_NumeroMesasDeseadas AT %DB9.DBW6, 100 ms
   "HMI_PiezaDisponiblesDeseadas" : Int = PLC HMI_vbes.HMI_NumeroMaterialesDeseados AT %DB9.DBW8, 100 ms
   "HMI_ReiniciarSistema" : Bool = PLC HMI_ReiniciarSistema AT %M12.2, 100 ms
   "HMI_vbes_HMI_ValorMesaSeleccionada" : Word = PLC HMI_vbes.HMI_ValorMesaSeleccionada AT %DB9.DBW2, 100 ms
   "HMI_vbes_HMI_MostrarPiezaE" : Bool = PLC HMI_vbes.HMI_MostrarPiezaE AT %DB9.DBX10.0, 100 ms
   "HMI_vbes_HMI_MostrarPiezaF" : Bool = PLC HMI_vbes.HMI_MostrarPiezaF AT %DB9.DBX10.1, 100 ms
   "HMI_vbes_HMI_MaterialDestino" : Word = PLC HMI_vbes.HMI_MaterialDestino AT %DB9.DBW12, 100 ms
   "HMI_vbes_HMI_MesaDestino" : Word = PLC HMI_vbes.HMI_MesaDestino AT %DB9.DBW14, 100 ms
   "HMI_vbes_HMI_Errores" : Word = PLC HMI_vbes.HMI_Errores AT %DB9.DBW16, 100 ms
   "HMI_vbes_HMI_MandarHome" : Bool = PLC HMI_vbes.HMI_MandarHome AT %DB9.DBX18.0, 100 ms
   "HMI_vbes_HMI_ApagarRobot" : Bool = PLC HMI_vbes.HMI_ApagarRobot AT %DB9.DBX18.1, 100 ms
   "HMI_vbes_HMI_PausarSistema" : Bool = PLC HMI_vbes.HMI_PausarSistema AT %DB9.DBX18.2, 100 ms

discrete alarms
   1: 'La instrucción enviada al robot no fue reconocida por el mismo', class Errors, trigger "HMI_vbes_HMI_Errores" bit 0
   2: 'El ID del material enviado al robot no es válido o no fue reconocido por el robot', class Errors, trigger "HMI_vbes_HMI_Errores" bit 1
   3: 'El número de mesa enviado al robot no es válido o no fue reconocido por el robot', class Errors, trigger "HMI_vbes_HMI_Errores" bit 2
   4: 'La longitud del mensaje enviado no es correcta', class Errors, trigger "HMI_vbes_HMI_Errores" bit 3
   5: 'El robot se ha desconectado', class Errors, trigger "HMI_vbes_HMI_Errores" bit 4
   6: 'El robot ha tenido un fallo fatal y deberá ser rearmado', class Errors, trigger "HMI_vbes_HMI_Errores" bit 5
   7: 'Error de numero de componentes por bandeja enviado en la configuración al robot', class Errors, trigger "HMI_vbes_HMI_Errores" bit 6
   8: 'Error de numero de mesas enviado en la configuración al robot', class Errors, trigger "HMI_vbes_HMI_Errores" bit 7
   9: 'El sensor de material del robot ha fallado mientras transportaba material.', class Errors, trigger "HMI_vbes_HMI_Errores" bit 8

text list "BotonFijar": 0 'Fijar'; 1 'Liberar'

text list "ListaMesas": 0 'Mesa 0'; 1 'Mesa 1'; 2 'Mesa 2'; 3 'Mesa 3'; 4 'Mesa 4'; 5 'Mesa 5'; 6 'Mesa 6'; 7 'Mesa 7'; 8 'Mesa 8'; 9 'Mesa 9'; 10 'Mesa 10'; 11 'Mesa 11'; 12 'Mesa 12'

text list "PausarSistema": 0 'Pausar'; 1 'Reanudar'

graphic list "CintaGeneralFlecha": 0 'CintaGeneral_OFF'; 1 'CintaGeneral_ON'

graphic list "CintaEmpaqFlecha": 0 'CintaEmp_OFF'; 1 'CintaEmp_ON'

graphic list "CintaA": 0 'FlechaCinta_OFF'; 1 'FlechaCinta_AMARILLO'

graphic list "CintaB": 0 'FlechaCinta_OFF'; 1 'FlechaCinta_VERDE'

graphic list "CintaC": 0 'FlechaCinta_OFF'; 1 'FlechaCinta_AZUL'

graphic list "CintaD": 0 'FlechaCinta_OFF'; 1 'FlechaCinta_ROJO'

graphic list "PaleE": 0 'PaleOFF'; 1 'PaleE'

graphic list "PaleF": 0 'PaleOFF'; 1 'PaleF'

graphic list "SP_I": 0 'SP_OFF'; 1 'SP_ON'

graphic list "SP_D": 0 'SP_OFF_D'; 1 'SP_ON_D'

graphic list "SP_A": 0 'SP_OFF_U'; 1 'SP_ON_U'

screen "Root screen" 1280x740, template "TemplateHome"
   on GenerateScreen: SetTag("Tag_ScreenNumber", 1); "IniciarBotonesMesas"()
   Button "Button_1" at 384,302 size 533x101; TextOff 'Iniciar'
      on Click: ActivateScreen("Pantalla Real", 0)

Template "TemplateHome" 1280x740
   Button "Alarms" at 1,3 size 78x59; TextOff 'Alarms'; PictureOff "AlarmDisplay_TP1200_Comfort_TR"; PictureOn "AlarmDisplay_TP1200_Comfort_TR"
      on Release: function_ef3f5d25("Alarm window_Unacknowledged", -1)
   Button "Template_Button" at 1,64 size 78x59; TextOff 'Text'
   Button "Template_Button_1" at 1,126 size 78x59; TextOff 'Text'
   Button "Template_Button_2" at 1,187 size 78x59; TextOff 'Text'
   Button "Template_Button_3" at 1,249 size 78x59; TextOff 'Text'
   Button "Template_Button_4" at 1,310 size 78x59; TextOff 'Text'
   Button "Template_Button_5" at 1,372 size 78x59; TextOff 'Text'
   Button "Template_Button_6" at 1,433 size 78x59; TextOff 'Text'
   Button "Template_Button_7" at 1,495 size 78x59; TextOff 'Text'
   Button "Template_Button_8" at 1,556 size 78x59; TextOff 'Text'
   Button "Template_Button_9" at 1,618 size 78x59; TextOff 'Text'
   Button "Template_Button_10" at 1,679 size 78x59; TextOff 'Text'

screen "System screens" 1280x740, template "TemplateHome"
   on GenerateScreen: SetTag("Tag_ScreenNumber", 2)
   Button "Back" at 80,1 size 159x47; TextOff 'Back'
      on Release: ActivateScreen("Root screen", 0)
   Button "HmiScreenItemData" at 115,95 size 159x47; TextOff 'SIMATIC PLC system diagnos...'; PictureOff "Navigates to SIMATIC PLC system diagnostics for TP1200 Comfort 17.0.0.0"; PictureOn "Navigates to SIMATIC PLC system diagnostics for TP1200 Comfort 17.0.0.0"
      on Release: ActivateScreen("SIMATIC PLC system diagnostics", 0)
   Button "HmiScreenItemData_1" at 115,154 size 159x47; TextOff 'Project information'; PictureOff "Navigates to Project information for TP1200 Comfort 17.0.0.0"; PictureOn "Navigates to Project information for TP1200 Comfort 17.0.0.0"
      on Release: ActivateScreen("Project information", 0)
   Button "HmiScreenItemData_2" at 115,213 size 159x47; TextOff 'System settings'; PictureOff "Navigates to System settings for TP1200 Comfort 17.0.0.0"; PictureOn "Navigates to System settings for TP1200 Comfort 17.0.0.0"
      on Release: ActivateScreen("System settings", 0)
   Button "HmiScreenItemData_3" at 115,272 size 159x47; TextOff 'User administration'; PictureOff "Navigates to User administration for TP1200 Comfort 17.0.0.0"; PictureOn "Navigates to User administration for TP1200 Comfort 17.0.0.0"
      on Release: ActivateScreen("User administration", 0)
   Button "HmiScreenItemData_4" at 115,331 size 159x47; TextOff 'System information'; PictureOff "Navigates to System information for TP1200 Comfort 17.0.0.0"; PictureOn "Navigates to System information for TP1200 Comfort 17.0.0.0"
      on Release: ActivateScreen("System information", 0)
   Button "HmiScreenItemData_5" at 115,390 size 159x47; TextOff 'Different jobs'; PictureOff "Navigates to Different jobs for TP1200 Comfort 17.0.0.0"; PictureOn "Navigates to Different jobs for TP1200 Comfort 17.0.0.0"
      on Release: ActivateScreen("Different jobs", 0)

screen "SIMATIC PLC system diagnostics" 1280x740, template "TemplateHome"
   on GenerateScreen: SetTag("Tag_ScreenNumber", 3)
   SysDiagControl "HmiScreenItemData" at 80,49 size 1197x683
   Button "Back" at 80,1 size 159x47; TextOff 'Back'
      on Release: ActivateScreen("System screens", 0)

screen "Project information" 1280x740, template "TemplateHome"
   on GenerateScreen: SetTag("Tag_ScreenNumber", 4)
   TextField "HmiScreenItemData" at 114,51 size 171x28; Text 'Project name:'
   TextField "HmiScreenItemData_1" at 320,51 size 925x28; Text 'TFM_DanielBejar_S71500'
   TextField "HmiScreenItemData_2" at 114,81 size 171x28; Text 'Created on:'
   TextField "HmiScreenItemData_3" at 320,81 size 925x28; Text '6/3/2024 7:42:33 PM'
   TextField "HmiScreenItemData_4" at 114,111 size 171x28; Text 'Author:'
   TextField "HmiScreenItemData_5" at 320,111 size 925x28; Text 'Daniel'
   TextField "HmiScreenItemData_6" at 114,141 size 171x28; Text 'Description:'
   TextField "HmiScreenItemData_7" at 320,141 size 925x28; Text '(not configured)'
   Button "Back" at 80,1 size 159x47; TextOff 'Back'
      on Release: ActivateScreen("System screens", 0)

screen "System settings" 1280x740, template "TemplateHome"
   on GenerateScreen: SetTag("Tag_ScreenNumber", 5)
   Button "Calibrate screen" at 115,95 size 159x47; TextOff 'Calibrate screen'
      on Release: function_bc3e350c()
   Button "Clean screen" at 115,154 size 159x47; TextOff 'Clean screen'
      on Release: function_be740847(30)
   Button "Back" at 80,1 size 159x47; TextOff 'Back'
      on Release: ActivateScreen("System screens", 0)

screen "User administration" 1280x740, template "TemplateHome"
   on GenerateScreen: SetTag("Tag_ScreenNumber", 6)
   UserView "HmiScreenItemData" at 80,49 size 1197x683
   Button "Back" at 80,1 size 159x47; TextOff 'Back'
      on Release: ActivateScreen("System screens", 0)

screen "System information" 1280x740, template "TemplateHome"
   on GenerateScreen: SetTag("Tag_ScreenNumber", 7)
   TextField "HmiScreenItemData" at 114,51 size 171x28; Text 'HMI device type:'
   TextField "HmiScreenItemData_1" at 320,51 size 925x28; Text 'TP1200 Comfort 17.0.0.0'
   TextField "HmiScreenItemData_2" at 114,81 size 171x28; Text 'Version:'
   TextField "HmiScreenItemData_3" at 114,111 size 171x28; Text 'Connection:'
   TextField "HmiScreenItemData_4" at 320,111 size 925x28; Text 'ETHERNET'
   TextField "HmiScreenItemData_5" at 114,141 size 171x28; Text 'PLC:'
   TextField "HmiScreenItemData_6" at 320,141 size 925x28; Text 'SIMATIC S7 1500'
   Button "Display version" at 320,81 size 925x28; TextOff 'Display version'
      on Release: function_febcb963(-1)
   Button "Back" at 80,1 size 159x47; TextOff 'Back'
      on Release: ActivateScreen("System screens", 0)

screen "Different jobs" 1280x740, template "TemplateHome"
   on GenerateScreen: SetTag("Tag_ScreenNumber", 8)
   Button "Online" at 115,95 size 159x47; TextOff 'Online'
      on Release: function_bb44b551(0)
   Button "Offline" at 115,154 size 159x47; TextOff 'Offline'
      on Release: function_bb44b551(1)
   Button "Transfer" at 115,213 size 159x47; TextOff 'Transfer'
      on Release: function_bb44b551(2)
   Button "Toggle language" at 115,272 size 159x47; TextOff 'Toggle language'
      on Release: function_fb9197e8(-1)
   Button "Control Panel" at 115,331 size 159x47; TextOff 'Control Panel'
      on Release: function_f34a74f3()
   Button "Stop Runtime" at 115,390 size 159x47; TextOff 'Stop Runtime'
      on Release: StopRuntime(0)
   Button "Back" at 80,1 size 159x47; TextOff 'Back'
      on Release: ActivateScreen("System screens", 0)

screen "Pantalla Simulacion" 1280x740, template "TemplateOtra"
   on GenerateScreen: SetTag("Tag_ScreenNumber", 20); "IniciarBotonesMesas"()
   Button "HmiScreenItemData_1" at 104,674 size 146x47; TextOn 'System screens'; TextOff 'System screens'; PictureOn "Navigates to System screens for TP1200 Comfort 17.0.0.0"; PictureOff "Navigates to System screens for TP1200 Comfort 17.0.0.0"
      on Release: ActivateScreen("System screens", 0)
   GraphicView "Graphic view_1" at 103,0 size 1144x740; Picture "FondoPrincipal_2"
   GraphicIOField "Graphic I/O field_1" at 151,395 size 636x57; PictureList "CintaGeneralFlecha"
      ProcessValue <- "CintaGeneral"
   GraphicIOField "Graphic I/O field_2" at 801,526 size 51x191; PictureList "CintaEmpaqFlecha"
      ProcessValue <- "CintaEmpaquetado"
   Circle "Circle_1" at 870,418 size 25x25
      Appearance <- "vbes_RobotConectado"
   Circle "Circle_2" at 870,450 size 25x25
      Appearance <- "vbes_RobotOcupado"
   Button "CambiarModoSim" at 274,674 size 147x47; TextOff 'Modo real'
      on Click: ResetBit("vbes_ModoSimulacion"); ActivateScreen("Root screen", 0)
   Button "Button_9" at 733,202 size 65x32; TextOff 'Fijar'; TextList "BotonFijar"
      ProcessValue <- "SP_CintaGeneral_Forzado"
      on Click: InvertBit("SP_CintaGeneral_Forzado"); InvertBit("HMI_SP_CintaGeneral")
   Button "Button_10" at 1023,601 size 65x32; TextOff 'Fijar'; TextList "BotonFijar"
      on Click: InvertBit("SP_CintaEmpaq_Forzado"); InvertBit("HMI_SP_CintaEmpaquetado")
      ProcessValue <- "SP_CintaEmpaq_Forzado"
   Button "Button_1" at 174,83 size 52x175; TextOff 'Text'; PictureList "CintaA"
      on Click: function_c82f6f27("HMI_SP_Cintas", 0)
      ProcessValue <- "HMI_SP_Cintas"
   Button "Button_2" at 316,83 size 52x175; TextOff 'Text'; PictureList "CintaB"
      on Click: function_c82f6f27("HMI_SP_Cintas", 1)
      ProcessValue <- "HMI_SP_Cintas"
   Button "Button_3" at 461,83 size 52x175; TextOff 'Text'; PictureList "CintaC"
      on Click: function_c82f6f27("HMI_SP_Cintas", 2)
      ProcessValue <- "HMI_SP_Cintas"
   Button "Button_4" at 602,83 size 52x175; TextOff 'Text'; PictureList "CintaD"
      on Click: function_c82f6f27("HMI_SP_Cintas", 3); function_c82f6f27("HMI_SP_Cintas", 4)
      ProcessValue <- "HMI_SP_Cintas"
   Button "Button_5" at 832,35 size 63x63; TextOff 'Text'; PictureList "PaleE"
      ProcessValue <- "HMI_PaleE"
      on Click: InvertBit("HMI_PaleE")
   Button "Button_6" at 1003,35 size 63x63; TextOff 'Text'; PictureList "PaleF"
      on Click: InvertBit("HMI_PaleF")
      ProcessValue <- "HMI_PaleF"
   Button "Button_7" at 734,240 size 63x33; TextOff 'Text'; PictureOn "SP_ON_U"; PictureOff "SP_OFF_U"
      Visibility <- "SP_CintaGeneral"
      on Release: ResetBit("HMI_SP_CintaGeneral")
      on Press: SetBit("HMI_SP_CintaGeneral")
   GraphicView "Graphic view_7" at 734,239 size 63x33; Picture "SP_ON_U"
      Visibility <- "SP_CintaGeneral_Forzado"
   Button "Button_8" at 1033,526 size 33x63; TextOff 'Text'; PictureOn "SP_ON_D"; PictureOff "SP_OFF_D"
      Visibility <- "SP_CintaGeneral"
      on Press: SetBit("HMI_SP_CintaEmpaquetado")
      on Release: ResetBit("HMI_SP_CintaEmpaquetado")
   GraphicView "Graphic view_8" at 1033,527 size 33x63; Picture "SP_ON_D"
      Visibility <- "SP_CintaEmpaq_Forzado"
   Button "BotonMesa_0" at 1097,184 size 55x63; TextOff 'M0'
      on Click: "FuncBotonMesa"()
      Appearance <- "HMI_vbes_HMI_MesaDestino"
   Button "BotonMesa_1" at 1097,258 size 55x63; TextOff 'M1'
      on Click: "FuncBotonMesa"()
      Appearance <- "HMI_vbes_HMI_MesaDestino"
   Button "BotonMesa_2" at 1097,332 size 55x63; TextOff 'M2'
      on Click: "FuncBotonMesa"()
      Appearance <- "HMI_vbes_HMI_MesaDestino"
   Button "BotonMesa_3" at 1097,406 size 55x63; TextOff 'M3'
      on Click: "FuncBotonMesa"()
      Appearance <- "HMI_vbes_HMI_MesaDestino"
   Button "BotonMesa_4" at 1097,480 size 55x63; TextOff 'M4'
      on Click: "FuncBotonMesa"()
      Appearance <- "HMI_vbes_HMI_MesaDestino"
   Button "BotonMesa_5" at 1097,554 size 55x63; TextOff 'M5'
      on Click: "FuncBotonMesa"()
      Appearance <- "HMI_vbes_HMI_MesaDestino"
   Button "BotonMesa_6" at 1172,184 size 55x63; TextOff 'M6'
      on Click: "FuncBotonMesa"()
      Appearance <- "HMI_vbes_HMI_MesaDestino"
   Button "BotonMesa_7" at 1172,258 size 55x63; TextOff 'M7'
      on Click: "FuncBotonMesa"()
      Appearance <- "HMI_vbes_HMI_MesaDestino"
   Button "BotonMesa_8" at 1172,332 size 55x63; TextOff 'M8'
      on Click: "FuncBotonMesa"()
      Appearance <- "HMI_vbes_HMI_MesaDestino"
   Button "BotonMesa_9" at 1172,406 size 55x63; TextOff 'M9'
      on Click: "FuncBotonMesa"()
      Appearance <- "HMI_vbes_HMI_MesaDestino"
   Button "BotonMesa_10" at 1172,480 size 55x63; TextOff 'M10'
      on Click: "FuncBotonMesa"()
      Appearance <- "HMI_vbes_HMI_MesaDestino"
   Button "BotonMesa_11" at 1172,554 size 55x63; TextOff 'M11'
      on Click: "FuncBotonMesa"()
      Appearance <- "HMI_vbes_HMI_MesaDestino"
   Button "CambiarModoSim_1" at 490,674 size 147x47; TextOff 'Configuración'
      on Click: ActivateScreen("Pantalla Configuracion", 0)
   Button "Button_11" at 92,9 size 56x56; TextOff 'Text'; PictureOff "Atras"
      on Click: function_efd93a16()
   Button "Button_12" at 930,456 size 32x33; TextOff 'Text'; PictureOff "Home_1"
      on Click: SetBit("HMI_vbes_HMI_MandarHome")
      Visibility <- "vbes_RobotConectado"
   Button "Button_13" at 984,456 size 32x33; TextOff 'Text'; PictureOff "OnOff"
      on Click: SetBit("HMI_vbes_HMI_ApagarRobot")
      Visibility <- "vbes_RobotConectado"
   Button "CambiarModoSim_2" at 1091,670 size 147x47; TextOff 'Pausar'; TextList "PausarSistema"
      ProcessValue <- "HMI_vbes_HMI_PausarSistema"
      Appearance <- "HMI_vbes_HMI_PausarSistema"
      on Click: InvertBit("HMI_vbes_HMI_PausarSistema")
   TextField "Text field_1" at 820,417 size 45x25; Text 'CON'
   TextField "Text field_2" at 809,449 size 56x25; Text 'BUSY'
   TextField "Text field_3" at 186,216 size 29x31; Text 'A'
   TextField "Text field_4" at 327,216 size 29x31; Text 'B'
   TextField "Text field_5" at 470,216 size 29x31; Text 'C'
   TextField "Text field_6" at 613,216 size 29x31; Text 'D'
   TextField "Text field_7" at 1019,51 size 29x31; Text 'F'
   TextField "Text field_8" at 849,51 size 29x31; Text 'E'
   GraphicView "Graphic view_2" at 187,309 size 96x48; Picture "MatA"
      Visibility <- "HMI_vbes_HMI_MaterialDestino"
   GraphicView "Graphic view_3" at 330,309 size 96x48; Picture "MatB"
      Visibility <- "HMI_vbes_HMI_MaterialDestino"
   GraphicView "Graphic view_4" at 474,309 size 96x48; Picture "MatC"
      Visibility <- "HMI_vbes_HMI_MaterialDestino"
   GraphicView "Graphic view_5" at 617,309 size 96x48; Picture "MatD"
      Visibility <- "vbes_Material_Destino"
   GraphicView "Graphic view_6" at 617,309 size 96x48; Picture "MatD"
      Visibility <- "HMI_vbes_HMI_MaterialDestino"
   GraphicView "Graphic view_9" at 836,115 size 59x85; Picture "MatE"
      Visibility <- "HMI_BaseSeleccionada"
   GraphicView "Graphic view_10" at 1007,115 size 59x85; Picture "MatF"
      Visibility <- "HMI_TapaSeleccionada"
   Rectangle "Rectangle_1" at 107,443 size 530x223
      Visibility <- "MesaSeleccionada"
   GraphicView "MaterialE" at 329,459 size 285x186; Picture "PiezaE"
      Visibility <- "HMI_vbes_HMI_MostrarPiezaE"
   GraphicView "MaterialA" at 341,468 size 152x99; Picture "PiezaA"
      Visibility <- "HMI_vbes_HMI_ValorMesaSeleccionada"
   GraphicView "MaterialB" at 341,552 size 71x78; Picture "PiezaB"
      Visibility <- "HMI_vbes_HMI_ValorMesaSeleccionada"
   GraphicView "MaterialC" at 422,552 size 71x78; Picture "PiezaC"
      Visibility <- "HMI_vbes_HMI_ValorMesaSeleccionada"
   GraphicView "MaterialD1" at 501,468 size 99x75; Picture "PiezaD"
      Visibility <- "HMI_vbes_HMI_ValorMesaSeleccionada"
   GraphicView "MaterialD2" at 502,553 size 99x75; Picture "PiezaD"
      Visibility <- "HMI_vbes_HMI_ValorMesaSeleccionada"
   GraphicView "MaterialF" at 321,451 size 304x207; Picture "PiezaF"
      Visibility <- "HMI_vbes_HMI_MostrarPiezaF"
   SymbolicIOField "Symbolic I/O field_1" at 129,471 size 169x48; TextOff '0'; TextOn '1'; TextList "ListaMesas"
      Visibility <- "MesaSeleccionada"
      ProcessValue <- "NumeroMesaSeleccionada"

screen "Pantalla Configuracion" 1280x740, template "TemplateOtra"
   IOField "I/O field_1" at 776,81 size 409x43; FormatPattern 99
      ProcessValue <- "HMI_MesasDisponiblesDeseadas"
   TextField "Text field_1" at 169,85 size 579x35; Text 'Número máximo de bandejas en paralelo'
   Button "Button_11" at 92,9 size 56x56; TextOff 'Text'; PictureOff "Atras"
      on Click: function_efd93a16()
   IOField "I/O field_2" at 776,145 size 409x43; FormatPattern 9
      ProcessValue <- "HMI_PiezaDisponiblesDeseadas"
   TextField "Text field_2" at 170,149 size 528x35; Text 'Número de componentes por bandeja'
   Button "Button_1" at 776,213 size 411x47; TextOff 'Reiniciar'; TextOn 'Reiniciando'
      on Press: SetBit("HMI_ReiniciarSistema")
      on Release: ResetBit("HMI_ReiniciarSistema")
   TextField "Text field_3" at 169,218 size 406x35; Text 'Reiniciar errores del sistema'

screen "Pantalla Real" 1280x740, template "TemplateOtra"
   on GenerateScreen: SetTag("Tag_ScreenNumber", 1); "IniciarBotonesMesas"()
   Button "HmiScreenItemData_1" at 104,674 size 146x47; TextOn 'System screens'; TextOff 'System screens'; PictureOn "Navigates to System screens for TP1200 Comfort 17.0.0.0"; PictureOff "Navigates to System screens for TP1200 Comfort 17.0.0.0"
      on Release: ActivateScreen("System screens", 0)
   GraphicView "Graphic view_1" at 103,0 size 1144x740; Picture "FondoPrincipal_2"
   GraphicIOField "Graphic I/O field_1" at 151,395 size 636x57; PictureList "CintaGeneralFlecha"
      ProcessValue <- "CintaGeneral"
   GraphicIOField "Graphic I/O field_2" at 801,526 size 51x191; PictureList "CintaEmpaqFlecha"
      ProcessValue <- "CintaEmpaquetado"
   Circle "Circle_1" at 870,418 size 25x25
      Appearance <- "vbes_RobotConectado"
   Circle "Circle_2" at 870,450 size 25x25
      Appearance <- "vbes_RobotOcupado"
   Button "CambiarModoSim" at 274,674 size 147x47; TextOff 'Modo simulación'
      on Click: SetBit("vbes_ModoSimulacion"); ActivateScreen("Pantalla Simulacion", 0)
   Button "Button_11" at 92,9 size 56x56; TextOff 'Text'; PictureOff "Atras"
      on Click: function_efd93a16()
   Button "BotonMesa_0" at 1097,184 size 55x63; TextOff 'M0'
      on Click: "FuncBotonMesa"()
      Appearance <- "HMI_vbes_HMI_MesaDestino"
   Button "BotonMesa_1" at 1097,258 size 55x63; TextOff 'M1'
      on Click: "FuncBotonMesa"()
      Appearance <- "HMI_vbes_HMI_MesaDestino"
   Button "BotonMesa_2" at 1097,332 size 55x63; TextOff 'M2'
      on Click: "FuncBotonMesa"()
      Appearance <- "HMI_vbes_HMI_MesaDestino"
   Button "BotonMesa_3" at 1097,406 size 55x63; TextOff 'M3'
      on Click: "FuncBotonMesa"()
      Appearance <- "HMI_vbes_HMI_MesaDestino"
   Button "BotonMesa_4" at 1097,480 size 55x63; TextOff 'M4'
      on Click: "FuncBotonMesa"()
      Appearance <- "HMI_vbes_HMI_MesaDestino"
   Button "BotonMesa_5" at 1097,554 size 55x63; TextOff 'M5'
      on Click: "FuncBotonMesa"()
      Appearance <- "HMI_vbes_HMI_MesaDestino"
   Button "BotonMesa_6" at 1172,184 size 55x63; TextOff 'M6'
      on Click: "FuncBotonMesa"()
      Appearance <- "HMI_vbes_HMI_MesaDestino"
   Button "BotonMesa_7" at 1172,258 size 55x63; TextOff 'M7'
      on Click: "FuncBotonMesa"()
      Appearance <- "HMI_vbes_HMI_MesaDestino"
   Button "BotonMesa_8" at 1172,332 size 55x63; TextOff 'M8'
      on Click: "FuncBotonMesa"()
      Appearance <- "HMI_vbes_HMI_MesaDestino"
   Button "BotonMesa_9" at 1172,406 size 55x63; TextOff 'M9'
      on Click: "FuncBotonMesa"()
      Appearance <- "HMI_vbes_HMI_MesaDestino"
   Button "BotonMesa_10" at 1172,480 size 55x63; TextOff 'M10'
      on Click: "FuncBotonMesa"()
      Appearance <- "HMI_vbes_HMI_MesaDestino"
   Button "BotonMesa_11" at 1172,554 size 55x63; TextOff 'M11'
      on Click: "FuncBotonMesa"()
      Appearance <- "HMI_vbes_HMI_MesaDestino"
   Button "CambiarModoSim_1" at 490,674 size 147x47; TextOff 'Configuración'
      on Click: ActivateScreen("Pantalla Configuracion", 0)
   Button "Button_1" at 92,9 size 56x56; TextOff 'Text'; PictureOff "Atras"
      on Click: function_efd93a16()
   Button "Button_12" at 930,456 size 32x33; TextOff 'Text'; PictureOff "Home_1"
      on Click: SetBit("HMI_vbes_HMI_MandarHome")
      Visibility <- "vbes_RobotConectado"
   Button "Button_13" at 984,456 size 32x33; TextOff 'Text'; PictureOff "OnOff"
      on Click: SetBit("HMI_vbes_HMI_ApagarRobot")
      Visibility <- "vbes_RobotConectado"
   Button "CambiarModoSim_2" at 1091,670 size 147x47; TextOff 'Pausar'; TextList "PausarSistema"
      on Click: InvertBit("HMI_vbes_HMI_PausarSistema")
      Appearance <- "HMI_vbes_HMI_PausarSistema"
      ProcessValue <- "HMI_vbes_HMI_PausarSistema"
   TextField "Text field_1" at 820,417 size 45x25; Text 'CON'
   TextField "Text field_2" at 809,449 size 56x25; Text 'BUSY'
   TextField "Text field_3" at 186,216 size 29x31; Text 'A'
   TextField "Text field_4" at 327,216 size 29x31; Text 'B'
   TextField "Text field_5" at 470,216 size 29x31; Text 'C'
   TextField "Text field_6" at 613,216 size 29x31; Text 'D'
   TextField "Text field_7" at 1019,51 size 29x31; Text 'F'
   TextField "Text field_8" at 849,51 size 29x31; Text 'E'
   GraphicView "Graphic view_2" at 187,309 size 96x48; Picture "MatA"
      Visibility <- "vbes_Material_Destino"
   GraphicView "Graphic view_3" at 330,309 size 96x48; Picture "MatB"
      Visibility <- "vbes_Material_Destino"
   GraphicView "Graphic view_4" at 474,309 size 96x48; Picture "MatC"
      Visibility <- "vbes_Material_Destino"
   GraphicView "Graphic view_5" at 617,309 size 96x48; Picture "MatD"
      Visibility <- "vbes_Material_Destino"
   GraphicView "Graphic view_6" at 617,309 size 96x48; Picture "MatD"
      Visibility <- "vbes_Material_Destino"
   GraphicIOField "Graphic I/O field_3" at 115,225 size 27x52; PictureList "SP_I"
      ProcessValue <- "SP_Cintas"
   GraphicIOField "Graphic I/O field_4" at 259,225 size 27x52; PictureList "SP_I"
      ProcessValue <- "SP_Cintas"
   GraphicIOField "Graphic I/O field_5" at 402,225 size 27x52; PictureList "SP_I"
      ProcessValue <- "SP_Cintas"
   GraphicIOField "Graphic I/O field_6" at 548,225 size 27x52; PictureList "SP_I"
      ProcessValue <- "SP_Cintas"
   GraphicIOField "Graphic I/O field_7" at 756,41 size 27x52; PictureList "SP_I"
      ProcessValue <- "SP_Cintas"
   GraphicIOField "Graphic I/O field_8" at 1114,41 size 27x52; PictureList "SP_D"
      ProcessValue <- "SP_Cintas"
   GraphicIOField "Graphic I/O field_11" at 1039,510 size 27x52; PictureList "SP_D"
      ProcessValue <- "SP_CintaEmpaquetado"
   GraphicIOField "Graphic I/O field_9" at 174,83 size 52x175; PictureList "CintaA"
      ProcessValue <- "SP_Cintas"
   GraphicIOField "Graphic I/O field_10" at 316,83 size 52x175; PictureList "CintaA"
      ProcessValue <- "SP_Cintas"
   GraphicIOField "Graphic I/O field_12" at 461,83 size 52x175; PictureList "CintaA"
      ProcessValue <- "SP_Cintas"
   GraphicIOField "Graphic I/O field_13" at 602,83 size 52x175; PictureList "CintaA"
      ProcessValue <- "SP_Cintas"
   GraphicIOField "Graphic I/O field_14" at 602,83 size 52x175; PictureList "CintaA"
      Visibility <- "SP_Cintas"
      ProcessValue <- "SP_Cintas"
   GraphicIOField "Graphic I/O field_15" at 832,35 size 63x63; PictureList "PaleE"
      ProcessValue <- "SP_Cintas"
   GraphicIOField "Graphic I/O field_16" at 1003,35 size 63x63; PictureList "PaleF"
      ProcessValue <- "SP_Cintas"
   GraphicIOField "Graphic I/O field_17" at 738,243 size 63x33; PictureList "SP_A"
      ProcessValue <- "SP_CintaGeneral"
   Rectangle "Rectangle_1" at 107,443 size 530x223
      Visibility <- "MesaSeleccionada"
   GraphicView "MaterialE" at 329,459 size 285x186; Picture "PiezaE"
      Visibility <- "HMI_vbes_HMI_MostrarPiezaE"
   GraphicView "MaterialA" at 341,468 size 152x99; Picture "PiezaA"
      Visibility <- "HMI_vbes_HMI_ValorMesaSeleccionada"
   GraphicView "MaterialB" at 341,552 size 71x78; Picture "PiezaB"
      Visibility <- "HMI_vbes_HMI_ValorMesaSeleccionada"
   GraphicView "MaterialC" at 422,552 size 71x78; Picture "PiezaC"
      Visibility <- "HMI_vbes_HMI_ValorMesaSeleccionada"
   GraphicView "MaterialD1" at 501,468 size 99x75; Picture "PiezaD"
      Visibility <- "HMI_vbes_HMI_ValorMesaSeleccionada"
   GraphicView "MaterialD2" at 502,553 size 99x75; Picture "PiezaD"
      Visibility <- "HMI_vbes_HMI_ValorMesaSeleccionada"
   GraphicView "MaterialF" at 321,451 size 304x207; Picture "PiezaF"
      Visibility <- "HMI_vbes_HMI_MostrarPiezaF"
   SymbolicIOField "Symbolic I/O field_1" at 129,471 size 169x48; TextOn '1'; TextOff '0'; TextList "ListaMesas"
      ProcessValue <- "NumeroMesaSeleccionada"
      Visibility <- "MesaSeleccionada"

Template "TemplateOtra" 1280x740
   Button "Alarms" at 1,3 size 78x59; TextOn 'Alarms'; TextOff 'Alarms'; PictureOn "AlarmDisplay_TP1200_Comfort_TR"; PictureOff "AlarmDisplay_TP1200_Comfort_TR"
      on Release: function_ef3f5d25("Alarm window_Unacknowledged", -1)
   Button "Template_Button" at 1,64 size 78x59; TextOff 'Text'
   Button "Template_Button_1" at 1,126 size 78x59; TextOff 'Text'
   Button "Template_Button_2" at 1,187 size 78x59; TextOff 'Text'
   Button "Template_Button_3" at 1,249 size 78x59; TextOff 'Text'
   Button "Template_Button_4" at 1,310 size 78x59; TextOff 'Text'
   Button "Template_Button_5" at 1,372 size 78x59; TextOff 'Text'
   Button "Template_Button_6" at 1,433 size 78x59; TextOff 'Text'
   Button "Template_Button_7" at 1,495 size 78x59; TextOff 'Text'
   Button "Template_Button_8" at 1,556 size 78x59; TextOff 'Text'
   Button "Template_Button_9" at 1,618 size 78x59; TextOff 'Text'
   Button "Template_Button_10" at 1,679 size 78x59; TextOff 'Text'

VB script "FuncBotonMesa"
   'Tip:
   ' 1. Use the <CTRL+SPACE> or <CTRL+I> shortcut to open a list of all objects and functions
   ' 2. Write the code using the HMI Runtime object.
   '  Example: HmiRuntime.Screens("Screen_1").
   ' 3. Use the <CTRL+J> shortcut to create an object reference.
   'Write the code as of this position:
   
   Dim nombreBoton, numMesa, valorMesa
   
   SmartTags("MesaSeleccionada") = Not SmartTags("MesaSeleccionada")
   nombreBoton = HmiRuntime.ActiveScreen.ActiveScreenItem.ObjectName
   numMesa = Split(nombreBoton, "_")(1)
   SmartTags("NumeroMesaSeleccionada") = numMesa

VB script "IniciarBotonesMesas"
   'Tip:
   ' 1. Use the <CTRL+SPACE> or <CTRL+I> shortcut to open a list of all objects and functions
   ' 2. Write the code using the HMI Runtime object.
   '  Example: HmiRuntime.Screens("Screen_1").
   ' 3. Use the <CTRL+J> shortcut to create an object reference.
   'Write the code as of this position:
   
   Dim numMesas, i
   
   numMesas = SmartTags("vbes_NumeroMesas")
   For i = 0 To numMesas
   	HmiRuntime.ActiveScreen.ScreenItems("BotonMesa_" & i).Visible = True
   Next
   For i = numMesas To 12
   	HmiRuntime.ActiveScreen.ScreenItems("BotonMesa_" & i).Visible = False
   Next
   
   SmartTags("MesaSeleccionada") = False
   SmartTags("NumeroMesaSeleccionada") = 0
*)